# B&R Automation Studio project mappFramework (part 6)

#### HMIActions.st
```iecst
ACTION VC4_Init:

	brsmemset(ADR(HmiFile.Status.FifoSelect[0]), 0, SIZEOF(HmiFile.Status.FifoSelect));
	IF HmiFile.Parameters.Fifo.Enable THEN
		HmiFile.Status.FifoSelect[HmiFile.Parameters.Fifo.SelectedDevice] := 1;
	END_IF;

	HmiFile.Status.FIFOLayerStatus := HIDE;

END_ACTION

ACTION VC4_Cyclic:

	MpFileManagerUISys.MpLink := ADR(gMpLinkFileManagerUIFile);
	MpFileManagerUISys.UIConnect := ADR(MpFileManagerUIConnect);
	MpFileManagerUISys();

	FOR i := 0 TO ((SIZEOF(HmiFile.Status.FileNames)/SIZEOF(HmiFile.Status.FileNames[0])) - 1) DO
		HmiFile.Status.FileNames[i] := MpFileManagerUIConnect.File.List.Items[i].Name;

		// Time Stamp
		HmiFile.Status.TimeStamps[i] := DT_TO_STRING(MpFileManagerUIConnect.File.List.Items[i].LastModified);
		HmiFile.Status.TimeStamps[i] := RIGHT(HmiFile.Status.TimeStamps[i], 19);

		// File size
		HmiFile.Status.Size[i] := REAL_TO_STRING(UDINT_TO_REAL(MpFileManagerUIConnect.File.List.Items[i].Size) * 0.001);

		// Set image array based on item type
		IF MpFileManagerUIConnect.File.List.Items[i].IsFolder THEN
			HmiFile.Status.Type[i] := FOLDER;
		ELSIF NOT MpFileManagerUIConnect.File.List.Items[i].IsFolder AND MpFileManagerUIConnect.File.List.Items[i].IsSelected THEN
			HmiFile.Status.Type[i] := FILE_SELECTED;
		ELSE
			HmiFile.Status.Type[i] := FILE;
		END_IF

		// Fill file info string arrays
		IF MpFileManagerUIConnect.File.List.Items[i].IsFolder THEN
			HmiFile.Status.InfoFile.Type[i] := 'FOLDER';
		ELSE
			HmiFile.Status.InfoFile.Type[i] := 'FILE';
		END_IF
		IF MpFileManagerUIConnect.File.List.Items[i].IsSelected THEN
			HmiFile.Status.InfoFile.IsSelected[i] := '+';
		ELSE
			HmiFile.Status.InfoFile.IsSelected[i] := '-';
		END_IF

		// If file does not exist, clear objects
		IF HmiFile.Status.FileNames[i] = '' THEN
			HmiFile.Status.TimeStamps[i] := '';
			HmiFile.Status.Size[i] := '';
			HmiFile.Status.InfoFile.IsSelected[i] := '';
			HmiFile.Status.InfoFile.Type[i] := '';
		END_IF;

	END_FOR

	// Mutli selection
	IF (NOT MpFileManagerUIConnect.File.MultiSelect) THEN
		MpFileManagerUIConnect.File.List.Items[HmiFile.Status.SelectedIndex].IsSelected := TRUE;
	ELSIF (MpFileManagerUIConnect.File.MultiSelect) AND HmiFile.Commands.FileList.Clicked THEN
		MpFileManagerUIConnect.File.List.Items[HmiFile.Status.SelectedIndex].IsSelected := NOT MpFileManagerUIConnect.File.List.Items[HmiFile.Status.SelectedIndex].IsSelected;
	END_IF
	HmiFile.Commands.FileList.Clicked := FALSE;

	// Read currently selected device name for HMI
	IF (MpFileManagerUIConnect.DeviceList.SelectedIndex >= (SIZEOF(MpFileManagerUIConnect.DeviceList.DeviceNames) / SIZEOF(MpFileManagerUIConnect.DeviceList.DeviceNames[0]))) THEN
		MpFileManagerUIConnect.DeviceList.SelectedIndex := 0;
	END_IF
	HmiFile.Status.DeviceName := MpFileManagerUIConnect.DeviceList.DeviceNames[MpFileManagerUIConnect.DeviceList.SelectedIndex];

	// Read if current selected object is folder
	IF (HmiFile.Status.SelectedIndex >= (SIZEOF(MpFileManagerUIConnect.File.List.Items) / SIZEOF(MpFileManagerUIConnect.File.List.Items[0]))) THEN
		HmiFile.Status.SelectedIndex := 0;
	END_IF
	HmiFile.Status.IsFolder := MpFileManagerUIConnect.File.List.Items[HmiFile.Status.SelectedIndex].IsFolder;

	// Control the folder structure when entering and leaving folders
	IF (HmiFile.Commands.EnterFolder) AND MpFileManagerUIConnect.File.List.Items[HmiFile.Status.SelectedIndex].IsFolder THEN
		HmiFile.Commands.EnterFolder := FALSE;
		MpFileManagerUIConnect.File.EnterFolder := TRUE;
		FolderDepthCount := FolderDepthCount + 1;
	ELSE
		HmiFile.Commands.EnterFolder := FALSE;
	END_IF

	IF EDGEPOS(HmiFile.Commands.FolderUp) AND (HmiFile.Status.BackButton > 0) THEN
		HmiFile.Commands.FolderUp := FALSE;
		MpFileManagerUIConnect.File.FolderUp := TRUE;
		FolderDepthCount := FolderDepthCount - 1;
	END_IF

	HmiFile.Status.BackButton := (FolderDepthCount > 0);

	// File SelectedIndex manager
	IF HmiFile.Commands.FileList.PageUp THEN
		HmiFile.Commands.FileList.PageUp := FALSE;
		HmiFile.Status.SelectedIndex := 0;

	ELSIF HmiFile.Commands.FileList.PageDown THEN
		HmiFile.Commands.FileList.PageDown := FALSE;
		HmiFile.Status.SelectedIndex := ((SIZEOF(HmiFile.Status.FileNames)/SIZEOF(HmiFile.Status.FileNames[0])) - 1);

	ELSIF HmiFile.Commands.FileList.StepUp THEN
		HmiFile.Commands.FileList.StepUp := FALSE;
		IF HmiFile.Status.SelectedIndex <> 0 THEN
			HmiFile.Status.SelectedIndex := HmiFile.Status.SelectedIndex - 1;
		END_IF

	ELSIF HmiFile.Commands.FileList.StepDown THEN
		HmiFile.Commands.FileList.StepDown := FALSE;
		IF HmiFile.Status.SelectedIndex <> ((SIZEOF(HmiFile.Status.FileNames)/SIZEOF(HmiFile.Status.FileNames[0])) - 1) THEN
			HmiFile.Status.SelectedIndex := HmiFile.Status.SelectedIndex + 1;
		END_IF
	END_IF

	HmiFile.Status.DefaultFileSelected := ((MpFileManagerUIConnect.File.List.Items[HmiFile.Status.SelectedIndex].Name = 'Default.par') OR
		(MpFileManagerUIConnect.File.List.Items[HmiFile.Status.SelectedIndex].Name = 'Machine.mcfg')) AND
		MpFileManagerUIConnect.DeviceList.SelectedIndex = 0;

END_ACTION

ACTION FormatDeviceDataProvider:

	// Select CF device if USB device is not available
	FOR i := 0 TO IDX_USB_DEV_LIST DO
		tempIdx := (i + USBOffset);

		IF gUSBAvailable[i] THEN
			PathCheck.DeviceList.DeviceNames[tempIdx] := 'USB';
			brsitoa(i + 1, ADR(PathCheck.DeviceList.DeviceNames[tempIdx]) + brsstrlen(ADR(PathCheck.DeviceList.DeviceNames[tempIdx])));
		ELSE
			brsmemset(ADR(HmiFile.Status.DeviceDataProvider[tempIdx]), 0, SIZEOF(HmiFile.Status.DeviceDataProvider[tempIdx]));
			brsmemset(ADR(PathCheck.DeviceList.DeviceNames[tempIdx]), 0, SIZEOF(PathCheck.DeviceList.DeviceNames[tempIdx]));
		END_IF
	END_FOR

	MaxDeviceNameIndex := ((SIZEOF(MpFileManagerUIConnect.DeviceList.DeviceNames) / SIZEOF(MpFileManagerUIConnect.DeviceList.DeviceNames[0])) - 1);
	// Check initilized folder for existance and remove any from the device list that don't exist
	IF (IdentStatus = 0) THEN
		// Copy device name from source list into the actual device list
		MpFileManagerUIConnect.DeviceList.DeviceNames[Index] := PathCheck.DeviceList.DeviceNames[DeviceListCount];
		Index := Index + 1;
		DeviceListCount := DeviceListCount + 1;

		IF (DeviceListCount > ((SIZEOF(PathCheck.DeviceList.DeviceNames) / SIZEOF(PathCheck.DeviceList.DeviceNames[0])) - 1)) THEN
			DeviceListCount := 0;
		END_IF
		IF (Index > MaxDeviceNameIndex) THEN
			Index := 0;
		END_IF
	ELSIF (IdentStatus = 3324) THEN
		DeviceListCount := DeviceListCount + 1;
		IF DeviceListCount > ((SIZEOF(PathCheck.DeviceList.DeviceNames) / SIZEOF(PathCheck.DeviceList.DeviceNames[0])) - 1) THEN
			// Delete entries past the actual number of devices found
			FOR i:=Index TO MaxDeviceNameIndex DO
				MpFileManagerUIConnect.DeviceList.DeviceNames[i] := '';
			END_FOR
			DeviceListCount := 0;
			Index := 0;
		END_IF
	END_IF

	IdentStatus := ST_ident(ADR(PathCheck.PrgName[DeviceListCount]),0,ADR(Ident));

	// Create device data provider for FIFO drop down
	FOR i := 0 TO MaxDeviceNameIndex DO
		IF (MpFileManagerUIConnect.DeviceList.DeviceNames[i] <> '') THEN
			HmiFile.Status.DeviceDataProvider[i] := MpFileManagerUIConnect.DeviceList.DeviceNames[i];
		ELSE
			brsmemset(ADR(HmiFile.Status.DeviceDataProvider[i]), 0, SIZEOF(HmiFile.Status.DeviceDataProvider[i]));
		END_IF
	END_FOR

END_ACTION
```

### Package Logical/Infrastructure/VC4/Usb - Package for USB handling for mapp Framework

### Program Logical/Infrastructure/VC4/Usb/UsbMgr (IEC) - Sample for all AsUSB-Library-Functions

#### UsbMgr.st - Cyclic code
```iecst
//*********************************************************************************
// Copyright: B&R Industrial Automation GmbH
// Author: B&R Industrial Automation GmbH
// Created: April 12, 2022
// Description: This task automatically detects and (un)links USB storage devices
//*********************************************************************************

PROGRAM _INIT
END_PROGRAM

PROGRAM _CYCLIC

	CASE StateMachine OF
		// -----------------------------------------------------------------------------------------------------------
		// Wait state
		// -----------------------------------------------------------------------------------------------------------
		USB_WAIT:
			// Refresh USB data every X seconds when enabled
			Node := 1;
			USB.Status := ERR_OK;
			IF USB.Cmd.AutoScan THEN
				RefreshTimer(IN := 1, PT := USB.Par.RefreshInterval);
				// Get new USB data
				IF(RefreshTimer.Q) THEN
					RefreshTimer(IN := 0);
					USB.Status := ERR_FUB_BUSY;
					brsmemset(ADR(UsbData), 0, SIZEOF(UsbData));
					StateMachine := USB_CREATE_NODE_ID_LIST;
				END_IF
			ELSE
				RefreshTimer(IN := 0);
			END_IF
			// Refresh USB data every X seconds when enabled
			IF USB.Cmd.ErrorReset THEN
				StateMachine := USB_ERROR;
			END_IF

			FOR i := 0 TO IDX_USB_DEV_LIST DO
				gUSBAvailable[i] := USB.Par.IsConnected[i+1];
			END_FOR

			// -----------------------------------------------------------------------------------------------------------
			// Get USB device list
			// -----------------------------------------------------------------------------------------------------------
		USB_CREATE_NODE_ID_LIST:
			GetUsbNodeList.enable := 1;
			GetUsbNodeList.pBuffer := ADR(NodeIdBuffer);
			GetUsbNodeList.bufferSize := SIZEOF(NodeIdBuffer);
			GetUsbNodeList.filterInterfaceClass := asusb_CLASS_MASS_STORAGE;
			GetUsbNodeList.filterInterfaceSubClass := 0;
			GetUsbNodeList;

			// --------------------------------------------------------------------------------------------------------------------
			// Success
			IF GetUsbNodeList.status = 0 THEN
				StateMachine := USB_READ_DEVICE_DATA;
				Node := 1;
				// No USB devices found
			ELSIF GetUsbNodeList.status = asusbERR_USB_NOTFOUND THEN
				// Unlink old device if it is gone now otherwise wait for next round
				FOR i:=1 TO MAX_IDX_USB_DEV_LIST DO
					IF(USB.Par.IsConnected[i]) THEN
						Node := 1;
						StateMachine := USB_CHECK_LINKED;
						RETURN;
					END_IF
				END_FOR;
				StateMachine := USB_WAIT;
				// Error
			ELSIF GetUsbNodeList.status <> ERR_FUB_BUSY THEN
				USB.Status := GetUsbNodeList.status;
				USB.Err.State := StateMachine;
				IF GetUsbNodeList.status = asusbERR_BUFSIZE THEN
					USB.Err.Text := 'maximum number of devices reached';
				ELSE
					USB.Err.Text := 'error getting device list';
				END_IF;
				StateMachine := USB_ERROR;
			END_IF;
			// -----------------------------------------------------------------------------------------------------------
			// Get device information
			// -----------------------------------------------------------------------------------------------------------
		USB_READ_DEVICE_DATA:
			GetUsbNode.enable := 1;
			GetUsbNode.nodeId := NodeIdBuffer[Node];
			GetUsbNode.pBuffer := ADR(UsbData[Node]);
			GetUsbNode.bufferSize := SIZEOF (UsbData[Node]);
			GetUsbNode;

			// --------------------------------------------------------------------------------------------------------------------
			// Success
			IF GetUsbNode.status = 0 THEN
				// Make sure we have enough space to store USB data, proceed with next StateMachine when all devices are detetced
				IF (Node = GetUsbNodeList.listNodes) OR (Node = MAX_IDX_USB_DEV_LIST) THEN
					Node := 1;
					StateMachine := USB_CHECK_LINKED;
					// Get next USB device
				ELSE
					Node := Node + 1;
				END_IF;
				// Error
			ELSIF GetUsbNode.status <> ERR_FUB_BUSY THEN
				USB.Status := GetUsbNode.status;
				USB.Err.State := StateMachine;
				USB.Err.Text := 'error getting device data';
				StateMachine := USB_ERROR;
			END_IF;
			// -----------------------------------------------------------------------------------------------------------
			// Check if linked device are still present
			// -----------------------------------------------------------------------------------------------------------
		USB_CHECK_LINKED:
			// Proceed to new devices when last device was checked
			IF(Node > MAX_IDX_USB_DEV_LIST) THEN
				Node := 1;
				StateMachine := USB_LINK_NEW;
				RETURN;
			END_IF

			// -----------------------------------------------------------------------------------------------------------
			// Check if device is still active
			IsLinked := FALSE;
			FOR i:=1 TO MAX_IDX_USB_DEV_LIST DO
				// Compare old and new data
				IF(brsmemcmp(ADR(UsbDataOld[Node]), ADR(UsbData[i]), SIZEOF(UsbData[i])) = 0) AND
					((NOT USB.Par.IgnoreDongle) OR (USB.Par.IgnoreDongle AND UsbData[i].productId <> BrProductId AND UsbData[i].vendorId <> BrVendorId)) THEN
					// Clear data, mark as linked and EXIT loop
					brsmemset(ADR(UsbData[i]), 0, SIZEOF(UsbData[i]));
					IsLinked := TRUE;
					EXIT;
				END_IF
			END_FOR;

			// -----------------------------------------------------------------------------------------------------------
			// Find next linked device
			IF(IsLinked OR UsbDataOld[Node].interfaceClass = 0) THEN
				IF(Node < MAX_IDX_USB_DEV_LIST) THEN
					Node := Node + 1;
					WHILE(Node < MAX_IDX_USB_DEV_LIST AND UsbDataOld[Node].interfaceClass = 0) DO
						Node := Node + 1;
					END_WHILE;
					IF(Node = MAX_IDX_USB_DEV_LIST AND UsbDataOld[Node].interfaceClass = 0) THEN
						Node := Node + 1;
					END_IF
				ELSE
					Node := Node + 1;
				END_IF
				// Unlink device if it is missing
			ELSE
				StateMachine := USB_UNLINK_DEVICE;
			END_IF
			// -----------------------------------------------------------------------------------------------------------
			// Link new devices
			// -----------------------------------------------------------------------------------------------------------
		USB_LINK_NEW:
			// Return to wait state when last device was checked
			IF(Node > MAX_IDX_USB_DEV_LIST) THEN
				StateMachine := USB_WAIT;
				RETURN;
			END_IF

			// -----------------------------------------------------------------------------------------------------------
			// Find next new device
			IF(UsbData[Node].interfaceClass <> 0) THEN
				IF((NOT USB.Par.IgnoreDongle) OR (UsbData[Node].productId <> BrProductId AND UsbData[Node].vendorId <> BrVendorId)) THEN
					StateMachine := USB_LINK_DEVICE;
					RETURN;
				END_IF
			END_IF
			Node := Node + 1;
			// -----------------------------------------------------------------------------------------------------------
			// Link device
			// -----------------------------------------------------------------------------------------------------------
		USB_LINK_DEVICE:
			// Find empty slot
			FOR i:=1 TO MAX_IDX_USB_DEV_LIST DO
				IF(UsbDataOld[i].interfaceClass = 0) THEN
					EXIT;
				END_IF
			END_FOR;
			// No more slot available
			IF(i = MAX_IDX_USB_DEV_LIST AND UsbDataOld[i].interfaceClass <> 0) THEN
				USB.Status := ERR_MAX_DEVICE;
				USB.Err.State := StateMachine;
				USB.Err.Text := 'maximum number of device reached';
				StateMachine := USB_ERROR;
				RETURN;
			END_IF
			// Create device string
			brsstrcpy(ADR(DevicePara), ADR('/DEVICE='));
			brsstrcat(ADR(DevicePara), ADR(UsbData[Node].ifName));
			brsstrcpy(ADR(DeviceName), ADR('USB'));
			brsitoa(i, ADR(tmpSTR));
			brsstrcat(ADR(DeviceName), ADR(tmpSTR));
			// Link device
			DevLinkSys.enable := 1;
			DevLinkSys.pDevice := ADR(DeviceName);
			DevLinkSys.pParam := ADR(DevicePara);
			DevLinkSys;

			// --------------------------------------------------------------------------------------------------------------------
			// Success
			IF DevLinkSys.status = 0 THEN
				// Store data for new device
				brsmemcpy(ADR(UsbDataOld[i]), ADR(UsbData[Node]), SIZEOF(UsbData[Node]));
				USB.Par.IsConnected[i] := TRUE;
				LinkHandle[i] := DevLinkSys.handle;
				Node := Node + 1;
				StateMachine := USB_LINK_NEW;
				// Error
			ELSIF DevLinkSys.status <> ERR_FUB_BUSY THEN
				USB.Status := DevLinkSys.status;
				USB.Err.State := StateMachine;
				USB.Err.Text := 'error linking device';
				StateMachine := USB_ERROR;
			END_IF;
			// -----------------------------------------------------------------------------------------------------------
			// UnLink device
			// -----------------------------------------------------------------------------------------------------------
		USB_UNLINK_DEVICE:
			DevUnlinkSys.enable := 1;
			DevUnlinkSys.handle := LinkHandle[Node];
			DevUnlinkSys;

			// --------------------------------------------------------------------------------------------------------------------
			// Success
			IF DevUnlinkSys.status = 0 THEN
				// Clear data
				brsmemset(ADR(UsbDataOld[Node]), 0, SIZEOF(UsbDataOld[Node]));
				USB.Par.IsConnected[Node] := FALSE;
				LinkHandle[Node] := 0;
				// Find next linked device
				WHILE(Node < MAX_IDX_USB_DEV_LIST AND UsbDataOld[Node].interfaceClass = 0) DO
					Node := Node + 1;
				END_WHILE;
				IF(Node = MAX_IDX_USB_DEV_LIST AND UsbDataOld[Node].interfaceClass = 0) THEN
					Node := Node + 1;
				END_IF
				StateMachine := USB_CHECK_LINKED;
				// Error
			ELSIF DevUnlinkSys.status <> ERR_FUB_BUSY THEN
				// Clear data
				brsmemset(ADR(UsbDataOld[Node]), 0, SIZEOF(UsbDataOld[Node]));
				USB.Par.IsConnected[Node] := FALSE;
				LinkHandle[Node] := 0;

				brsitoa(Node, ADR(tmpSTR));
				USB.Status := DevUnlinkSys.status;
				USB.Err.State := StateMachine;
				USB.Err.Text := 'error unlinking device no ';
				brsstrcat(ADR(USB.Err.Text), ADR(tmpSTR));
				StateMachine := USB_ERROR;
			END_IF;
			// -----------------------------------------------------------------------------------------------------------
			// Error state
			// -----------------------------------------------------------------------------------------------------------
		USB_ERROR:
			// Get more error information
			IF(USB.Status = 0) THEN
				USB.Status := FileIoGetSysError();
			END_IF

			// Unlink device
			IF(USB.Err.State = USB_LINK_DEVICE) THEN
				DevUnlinkSys.enable := 1;
				DevUnlinkSys.handle := DevLinkSys.handle;
				DevUnlinkSys;
			END_IF

			// Reset error
			IF(USB.Cmd.ErrorReset AND DevUnlinkSys.status <> ERR_FUB_BUSY) THEN
				USB.Cmd.ErrorReset := FALSE;
				brsmemset(ADR(USB.Err), 0, SIZEOF(USB.Err));
				StateMachine := USB_WAIT;
			END_IF
	END_CASE;

END_PROGRAM

PROGRAM _EXIT
	FOR i:=1 TO MAX_IDX_USB_DEV_LIST DO
		REPEAT
			DevUnlinkSys.enable := 1;
			DevUnlinkSys.handle := LinkHandle[i];
			DevUnlinkSys;
			UNTIL DevUnlinkSys.status <> ERR_FUB_BUSY
		END_REPEAT;
	END_FOR;
END_PROGRAM
```

#### UsbMgr.typ - Local data types
```iecst
TYPE
	UsbStateEnum :
		(
		USB_WAIT, (*Wait for starting the Function chain*)
		USB_CREATE_NODE_ID_LIST, (*Create a list of Node-IDs from all active USB devices*)
		USB_READ_DEVICE_DATA, (*Read out the specific data from the Node-IDs*)
		USB_CHECK_LINKED, (*Check if device is still connected*)
		USB_LINK_NEW,
		USB_LINK_DEVICE, (*Link file device*)
		USB_UNLINK_DEVICE, (*Unlink the File Device from specific path*)
		USB_ERROR (*Jump to this step in every case of Error occuring in the Function chain*)
		);
	UsbCmdType : 	STRUCT
		AutoScan : BOOL := TRUE; (*Scan USB ports automatically*)
		ErrorReset : BOOL; (*Reset error*)
	END_STRUCT;
	UsbParType : 	STRUCT
		IgnoreDongle : BOOL := TRUE; (*Ignoe B&R license dongle*)
		RefreshInterval : TIME := T#3s; (*Intervall timer for USB device refresh*)
		IsConnected : ARRAY[0..MAX_IDX_USB_DEV_LIST]OF BOOL; (*Shows if a USB stick is connected*)
	END_STRUCT;
	UsbErrType : 	STRUCT
		State : UsbStateEnum; (*State where the error occured*)
		Text : STRING[80]; (*Error text*)
	END_STRUCT;
	UsbMainType : 	STRUCT
		Cmd : UsbCmdType; (*Command structure*)
		Par : UsbParType; (*Parameter structure*)
		Err : UsbErrType; (*Error structure*)
		Status : UINT; (*Current status*)
	END_STRUCT;
END_TYPE
```

#### UsbMgr.var - Local variables
```iecst
(*Function Blocks*)
VAR
	RefreshTimer : TON;
	GetUsbNodeList : UsbNodeListGet; (*Type of FUB UsbNodeListGet*)
	GetUsbNode : UsbNodeGet; (*Type of FUB UsbNodeGet*)
	DevLinkSys : DevLink; (*Type of FUB DevLink*)
	DevUnlinkSys : DevUnlink; (*Type of FUB DevUnlink*)
END_VAR
(*Constants*)
VAR CONSTANT
	BrVendorId : UINT := 1615; (*B&R vendor id*)
	BrProductId : UINT := 1001; (*B&R dongle product id*)
END_VAR
(*Structure Types*)
VAR
	USB : UsbMainType;
	StateMachine : UsbStateEnum; (*State machine*)
	UsbData : ARRAY[1..MAX_IDX_USB_DEV_LIST] OF usbNode_typ; (*Data of all available USB devices*)
	UsbDataOld : ARRAY[1..MAX_IDX_USB_DEV_LIST] OF usbNode_typ; (*Old data of all available USB devices*)
END_VAR
(*Variables*)
VAR
	DevicePara : STRING[80]; (*Connection path of USB device*)
	DeviceName : STRING[40]; (*Connection path of USB device*)
	LinkHandle : ARRAY[1..MAX_IDX_USB_DEV_LIST] OF UDINT; (*Link handle for USB device*)
	NodeIdBuffer : ARRAY[1..MAX_IDX_USB_DEV_LIST] OF UDINT; (*Different nodeIDs saved in array-elements*)
	IsLinked : BOOL; (*Helper variable that indicates that a USB stick is linked*)
	Node : USINT; (*Node number*)
	i : USINT;
	tmpSTR : STRING[10];
	ERR_MAX_DEVICE : UINT := 50000; (*Maximum number of dongles reached*)
END_VAR
```

### Package Logical/Infrastructure/VC4/Recipe - Package for mapp Recipe Framework

### Program Logical/Infrastructure/VC4/Recipe/RecipeMgr (IEC)

#### RecipeMgr.st - Init, cyclic, exit code
```iecst
//***********************************************************************
// Copyright: B&R Industrial Automation GmbH
// Author: B&R Industrial Automation GmbH
// Created: Jan 1, 2022
// Description: Tasks for recipe control with VC4 front-end.
//***********************************************************************

PROGRAM _INIT

	// Create folder for this component on the user file device
	DirCreateRecipe(enable := TRUE, pDevice := ADR('mappRecipeFiles'), pName := ADR('/'));

	// Wait for DirCreate_0 to complete.
	WHILE (DirCreateRecipe.status = ERR_FUB_BUSY) DO
		DirCreateRecipe();
	END_WHILE

	// Check if folder already exist and if so disabled the function block call
	IF DirCreateRecipe.status = fiERR_DIR_ALREADY_EXIST OR (DirCreateRecipe.status = ERR_OK) THEN
		DirCreateRecipe(enable := FALSE);
	END_IF

	// Initialize mapp function blocks
	// By default, the Framework sets up an XML recipe system. To swtich to the CSV format, refer to the "Change Recipe Format"
	// page in the AS Help (GUID 2052b3a5-f59b-45f9-9fcd-3289c93401af)
	MpRecipeUISetup.Confirmation.RecipeDelete := TRUE;
	MpRecipeUISetup.RecipeListSize := 9;
	MpRecipeUISetup.RecipeListScrollWindow := 0;
	MpRecipeUISetup.AutoLoadHeader := TRUE;
	MpRecipeUIConnect.New.FileName := 'newRecipe';
	MpRecipeUIConnect.Recipe.Filter := '*par';
	MpRecipeUISys.MpLink := ADR(gMpLinkRecipeXml);
	MpRecipeUISys.Enable := TRUE;
	MpRecipeUISys.UIConnect := ADR(MpRecipeUIConnect);
	MpRecipeUISys.UISetup := MpRecipeUISetup;
	MpRecipeUISys();

	HmiRecipe.Parameters.Category := PARAMETERS_CATEGORY;
	HmiRecipe.Status.DeviceDataProvider[0] := '{"value":"mappRecipeFiles","text":"CF/PLC"}';
	HmiRecipe.Parameters.DeviceName := 'mappRecipeFiles';
	MpRecipeSys.MpLink := ADR(gMpLinkRecipeXml);
	MpRecipeSys.Enable := TRUE;
	MpRecipeSys.Category := ADR(HmiRecipe.Parameters.Category);
	MpRecipeSys.DeviceName := ADR(HmiRecipe.Parameters.DeviceName);
	MpRecipeSys.FileName := ADR(HmiRecipe.Parameters.FileName);
	MpRecipeSys.Header := ADR(Header);

	// Wait for MpRecipeSys to activate. This must be active before you can call the RegPar function blocks, which is below.
	WHILE NOT(MpRecipeSys.Active OR MpRecipeSys.Error) DO
		MpRecipeSys();
	END_WHILE

	// Register the preview variables to the recipe. These preview variables are a buffer between the recipe system and the
	// variables used at runtime on the machine (Parameters, MachineSettings). By using these preview variables, you can
	// preview and edit a recipe on the HMI without actually loading it to the machine. For more details, refer to the
	// "Recipe System Design" page in the AS Help (GUID 3ccd7409-0b52-4bbc-a93a-4010f6db414c).

	MpRecipeRegPar_PreviewPar.MpLink := ADR(gMpLinkRecipeXml);
	MpRecipeRegPar_PreviewPar.Enable := TRUE;
	MpRecipeRegPar_PreviewPar.PVName := ADR('RecipeMgr:ParametersPreview');
	MpRecipeRegPar_PreviewPar.Category := ADR(PARAMETERS_CATEGORY);
	MpRecipeRegPar_PreviewPar();

	MpRecipeRegPar_PreviewCfg.MpLink := ADR(gMpLinkRecipeXml);
	MpRecipeRegPar_PreviewCfg.Enable := TRUE;
	MpRecipeRegPar_PreviewCfg.PVName := ADR('RecipeMgr:MachineSettingsPreview');
	MpRecipeRegPar_PreviewCfg.Category := ADR(MACHINE_CONFIGURATION_CATEGORY);
	MpRecipeRegPar_PreviewCfg();

	// Wait for RegPar function blocks to activate. These must be active before you can load a recipe,
	// which is further down in the Initialization program.
	WHILE NOT(MpRecipeRegPar_PreviewPar.Active OR MpRecipeRegPar_PreviewPar.Error) DO
		MpRecipeRegPar_PreviewPar();
	END_WHILE
	WHILE NOT(MpRecipeRegPar_PreviewCfg.Active OR MpRecipeRegPar_PreviewCfg.Error) DO
		MpRecipeRegPar_PreviewCfg();
	END_WHILE

	// Load default Machine Settings recipe
	HmiRecipe.Parameters.Category := MACHINE_CONFIGURATION_CATEGORY;
	HmiRecipe.Parameters.FileName := DEFAULT_MACHINE_CONFIGURATION;
	brsstrcat(ADR(HmiRecipe.Parameters.FileName),ADR(MACHINE_CONFIG_FILE_EXTENSION));
	MpRecipeSys.Load := TRUE;
	WHILE NOT(MpRecipeSys.CommandDone OR MpRecipeSys.Error) DO
		MpRecipeSys();
	END_WHILE
	MachineSettings := MachineSettingsPreview;
	HmiRecipe.Status.LastLoadedConfigRecipe := DEFAULT_MACHINE_CONFIGURATION;
	brsstrcat(ADR(HmiRecipe.Status.LastLoadedConfigRecipe),ADR(MACHINE_CONFIG_FILE_EXTENSION));
	HmiRecipe.Status.ConfigRecipeLoaded := TRUE;

	// Check if the default machine settings recipe is missing
	IF MpRecipeSys.Info.Diag.StatusID.ID = mpRECIPE_ERR_LOAD_DATA THEN
		HmiRecipe.Status.MachineSettingsRecipeMissing := TRUE;
		HmiRecipe.Status.LastLoadedConfigRecipe := '';
		HmiRecipe.Status.ConfigRecipeLoaded := FALSE;
	END_IF

	MpRecipeSys.ErrorReset := MpRecipeSys.Error;
	MpRecipeSys.Load := FALSE;
	MpRecipeSys();

	// Load default Parameter recipe
	HmiRecipe.Parameters.Category := PARAMETERS_CATEGORY;
	HmiRecipe.Parameters.FileName := DEFAULT_PARAMETERS;
	brsstrcat(ADR(HmiRecipe.Parameters.FileName),ADR(PARAMETERS_FILE_EXTENSION));
	HmiRecipe.Status.PreviousRecipe := DEFAULT_PARAMETERS;
	MpRecipeSys.Load := TRUE;
	WHILE NOT(MpRecipeSys.CommandDone OR MpRecipeSys.Error) DO
		MpRecipeSys();
	END_WHILE
	Parameters := ParametersPreview;
	HmiRecipe.Status.LastLoadedProductRecipe := DEFAULT_PARAMETERS;
	brsstrcat(ADR(HmiRecipe.Status.LastLoadedProductRecipe),ADR(PARAMETERS_FILE_EXTENSION));
	HmiRecipe.Status.ProductRecipeLoaded := TRUE;

	// Check if the default parameters recipe is missing
	IF MpRecipeSys.Info.Diag.StatusID.ID = mpRECIPE_ERR_LOAD_DATA THEN
		HmiRecipe.Status.ParameterRecipeMissing := TRUE;
		HmiRecipe.Status.LastLoadedProductRecipe := '';
		HmiRecipe.Status.ProductRecipeLoaded := FALSE;
	END_IF

	MpRecipeSys.ErrorReset := MpRecipeSys.Error;
	MpRecipeSys.Load := FALSE;
	MpRecipeSys();

	// Trigger update notification so that the initial parameters are copied to the process
	MpRecipeSys.UpdateNotification := TRUE;

	// Init Filemanager for exporting/importing files
	MpFileManagerUIRecipe.Enable := TRUE;
	MpFileManagerUIRecipe.MpLink := ADR(gMpLinkFileManagerUIRecipe);
	MpFileManagerUIRecipe.UIConnect := ADR(MpFileManagerUIConnect);
	MpFileManagerUIRecipe.UISetup.FileListSize := SIZEOF(MpFileManagerUIConnect.File.List.Items) / SIZEOF(MpFileManagerUIConnect.File.List.Items[0]);
	MpFileManagerUIConnect.DeviceList.DeviceNames[0] := 'mappRecipeFiles';
	MpFileManagerUIConnect.DeviceList.DeviceNames[1] := '';
	MpFileManagerUIRecipe();

	HmiRecipe.Status.HMIcommand := REC_HMI_WAIT;

	VC4_Init;

END_PROGRAM

PROGRAM _CYCLIC

	// Call actions
	FormatDeviceDataProvider;
	LoadPreview;
	RecipeHMIcommands;
	LoadStatus;

	// Reset commands on MpRecipe FUB
	IF MpRecipeSys.CommandDone THEN
		MpRecipeSys.Load := FALSE;
		MpRecipeSys.Save := FALSE;
		// Set update notification for machine category
		IF ((brsstrcmp(ADR(HmiRecipe.Parameters.Category), ADR(MACHINE_CONFIGURATION_CATEGORY)) = 0) AND (MpRecipeSys.Save)) THEN
			MpRecipeSys.UpdateNotification := TRUE;
		ELSE
			MpRecipeSys.UpdateNotification := FALSE;
		END_IF
	END_IF

	// Error reset
	IF NOT MpRecipeSys.Error THEN
		MpRecipeSys.ErrorReset := FALSE;
	END_IF

	IF NOT MpRecipeUISys.Error THEN
		MpRecipeUISys.ErrorReset := FALSE;
	END_IF

	// Assign MpLinks & address references
	MpRecipeSys.MpLink := ADR(gMpLinkRecipeXml);
	MpRecipeSys.DeviceName := ADR(HmiRecipe.Parameters.DeviceName);
	MpRecipeSys.Header := ADR(Header);
	MpRecipeUISys.MpLink := ADR(gMpLinkRecipeXml);
	MpRecipeUISys.UIConnect := ADR(MpRecipeUIConnect);
	MpFileManagerUIRecipe.MpLink := ADR(gMpLinkFileManagerUIRecipe);
	MpRecipeRegPar_PreviewPar.MpLink := ADR(gMpLinkRecipeXml);
	MpRecipeRegPar_PreviewPar.PVName := ADR('RecipeMgr:ParametersPreview');
	MpRecipeRegPar_PreviewPar.Category := ADR(PARAMETERS_CATEGORY);
	MpRecipeRegPar_PreviewCfg.MpLink := ADR(gMpLinkRecipeXml);
	MpRecipeRegPar_PreviewCfg.PVName := ADR('RecipeMgr:MachineSettingsPreview');
	MpRecipeRegPar_PreviewCfg.Category := ADR(MACHINE_CONFIGURATION_CATEGORY);
	MpFileManagerUIRecipe.UIConnect := ADR(MpFileManagerUIConnect);

	// Call function blocks
	MpRecipeSys();
	MpRecipeUISys();
	MpFileManagerUIRecipe();
	MpRecipeRegPar_PreviewPar();
	MpRecipeRegPar_PreviewCfg();

END_PROGRAM

PROGRAM _EXIT

	// Disable the function blocls to unlink the MpLinks
	MpRecipeSys.Enable := FALSE;
	MpRecipeUISys.Enable := FALSE;
	MpRecipeRegPar_PreviewPar.Enable := FALSE;
	MpRecipeRegPar_PreviewCfg.Enable := FALSE;
	MpFileManagerUIRecipe.Enable := FALSE;

	// Call function blocks
	MpRecipeSys();
	MpRecipeUISys();
	MpRecipeRegPar_PreviewPar();
	MpRecipeRegPar_PreviewCfg();
	MpFileManagerUIRecipe();

END_PROGRAM
```

#### RecipeMgr.typ - Local data types
```iecst
(*Structure types*)

TYPE
	RecipeHmiInterfaceType : 	STRUCT  (*Structure to hold commands, parameters and status from the HMI*)
		Commands : RecipeCommandsType; (*Structure to hold the commands from the HMI*)
		Parameters : RecipeParametersType; (*Structure to hold the parameters for the HMI*)
		Status : RecipeStatusType; (*Structure to hold status information from the mapp View HMI*)
	END_STRUCT;
	RecipeCommandsType : 	STRUCT  (*Structure to hold the commands from the HMI*)
		LoadRecipe : BOOL; (*Load recipe*)
		SaveSelectedRecipe : BOOL; (*Save the selected recipe (which is not necessarily the active recipe)*)
		CreateRecipe : BOOL; (*Create recipe*)
		ImportFromUSB : BOOL; (*Import from USB device*)
		ExportToUSB : BOOL; (*Export to USB device*)
		ResetPreview : BOOL; (*Reset the preview to empty/zeros in the event of an invalid recipe*)
	END_STRUCT;
	RecipeParametersType : 	STRUCT  (*Structure to hold the parameters for the HMI*)
		Category : STRING[30]; (*Current category*)
		CategoryIndex : USINT; (*Current category*)
		DeviceName : STRING[50]; (*Selected file device name*)
		FileName : STRING[255]; (*Recipe file name*)
	END_STRUCT;
	RecipeStatusType : 	STRUCT  (*Structure to hold status information from the mapp View HMI*)
		DefaultFilesDeleteButtonStatus : USINT;
		HMIcommand : RecipeHmiStepEnum; (*State machine step for HMI commands*)
		LastLoadedConfigRecipe : STRING[255]; (*Last loaded configuration recipe*)
		LastLoadedProductRecipe : STRING[255]; (*Last loaded product recipe*)
		ProductRecipeLoaded : BOOL; (*Product recipe was loaded*)
		ConfigRecipeLoaded : BOOL; (*Config recipe was loaded*)
		LastMaxSelection : UINT; (*The previous maximum number of recipes*)
		LastSelectedIndex : UINT; (*The previous selected index*)
		LastStatus : MpRecipeUIStatusEnum; (*The previous UI status*)
		EditDialogOpened : BOOL; (*Flag that the edit dialog box was opened*)
		CreateDialogOpened : BOOL; (*Flag that the create dialog box was opened*)
		PreviousRecipe : STRING[80]; (*Name of the previous recipe*)
		FileDuplicate : BOOL; (*Recipe file already exists, warn the user.*)
		FilesAvailable : BOOL; (*Control access to widget when no files are available*)
		InvalidRecipe : BOOL; (*The selected recipe cannot be previewed*)
		LoadingRecipeList : BOOL; (*The recipe list is loading*)
		MachineSettingsRecipeMissing : BOOL; (*Flag for if the default machine settings recipe is not present*)
		ParameterRecipeMissing : BOOL; (*Flag for if the default parameters recipe is not present*)
		LoadAllowed : BOOL; (*Flag for whether you can load a recipe. Recipe must exist and be valid. *)
		DeviceDataProvider : ARRAY[0..MAX_IDX_FILE_DEV]OF STRING[100]; (*File device data provider*)
		SelectedRecipe : STRING[255]; (*The name of the selected recipe*)
		ActiveRecipe : STRING[255];
		DefaultRecipeLayer : RecipeStatusDefRecLayerType;
		CreateRecipeLayer : RecipeStatusCteateRecLayerType;
		PreviewRecipeLayer : RecipeStatusPreviewRecLayerType;
		RecipeLoadLayer : RecipeStatusRecipeLoadLayerType;
		EditRecipeLayer : RecipeStatusEditRecLayerType;
		DuplicateLayer : USINT;
		DeviceValid : BOOL; (*Flag for whether FileDevice is valid. Prevents user from being prompted to load default recipe.*)
		InvalidRecipeLayer : BOOL;
		DefaultFilesCannotBeDeleteLayer : USINT;
		RecipePageOpenedNow : BOOL;
		LoadPreviewAfterPageOpened : BOOL;
	END_STRUCT;
	RecipeStatusDefRecLayerType : 	STRUCT
		Status : USINT;
	END_STRUCT;
	RecipeStatusCteateRecLayerType : 	STRUCT
		ParsStatus : USINT;
		MachConfigStatus : USINT;
		FileNameInputActive : USINT;
	END_STRUCT;
	RecipeStatusPreviewRecLayerType : 	STRUCT
		ParsStatus : USINT;
		MachConfigStatus : USINT;
	END_STRUCT;
	RecipeStatusRecipeLoadLayerType : 	STRUCT
		Status : USINT;
	END_STRUCT;
	RecipeStatusEditRecLayerType : 	STRUCT
		ParsStatus : USINT;
		MachConfigStatus : USINT;
		Save : BOOL;
	END_STRUCT;
	ParametersType : 	STRUCT  (*Demo / starter structure for machine parameters*)
		AddParametersHere1 : BOOL; (*Add your parameteres here *)
		AddParametersHere2 : STRING[80]; (*Add your parameteres here *)
		AddParametersHere3 : REAL; (*Add your parameteres here *)
		AddParametersHere4 : REAL; (*Add your parameteres here *)
		AddParametersHere5 : REAL; (*Add your parameteres here *)
	END_STRUCT;
	MachineSettingsType : 	STRUCT  (*Demo / starter structure for machine configuration settings*)
		AddMachineSettingsHere1 : USINT; (*Add your settings here*)
		AddMachineSettingsHere2 : DINT; (*Add your settings here*)
		AddMachineSettingsHere3 : BOOL; (*Add your settings here*)
		AddMachineSettingsHere4 : REAL; (*Add your settings here*)
		AddMachineSettingsHere5 : UINT; (*Add your settings here*)
	END_STRUCT;
END_TYPE

(*Enumerations*)

TYPE
	RecipeHmiStepEnum :
		( (*State machine step for HMI commands*)
		REC_HMI_WAIT, (*Wait*)
		REC_HMI_LOAD, (*Load recipe*)
		REC_HMI_SAVE, (*Save recipe*)
		REC_HMI_CREATE, (*Create recipe*)
		REC_HMI_RESET_PREVIEW (*Reset the preview values to 0 / empty*)
		);
END_TYPE

(**)
```

#### RecipeMgr.var - Local variables
```iecst
(*Function Blocks*)
VAR
	MpRecipeSys : MpRecipeXml; (*MpRecipe instance*)
	MpRecipeRegPar_PreviewPar : MpRecipeRegPar; (*MpRecipeRegPar instance for ParametersPreview variable*)
	MpRecipeRegPar_PreviewCfg : MpRecipeRegPar; (*MpRecipeRegPar instance for MachineSettingsPreview*)
	MpRecipeUISys : MpRecipeUI; (*MpRecupeUI instance*)
	MpFileManagerUIRecipe : MpFileManagerUI; (*MpFileManagerUI instance*)
	DTGetTimeRecipe : DTGetTime; (*DTGetTime instance*)
	DirCreateRecipe : DirCreate; (*DirCreate instance*)
END_VAR
(*Constants*)
VAR CONSTANT
	MAX_IDX_FILE_DEV : USINT := MAX_IDX_USB_DEV_LIST + 1; (*Maximum number of  file devices *)
END_VAR
VAR
	PARAMETERS_RECIPE : STRING[50] := 'Parameters'; (*Value of the DropDownBox selection for the Parameters category*)
	MACHINE_CONFIGURATION_RECIPE : STRING[50] := 'Machine Configuration'; (*Value of the DropDownBox selection for the Machine Configuration category*)
END_VAR
(*Structure Types*)
VAR
	HmiRecipe : RecipeHmiInterfaceType; (*HMI interface structure*)
	Parameters : ParametersType; (*Machine parameters. Used by the machine at runtime*)
	ParametersEdit : {REDUND_UNREPLICABLE} ParametersType; (*Machine parameters edit structure. Enables you to edit a recipe that is not currently active*)
	ParametersPreview : ParametersType; (*Machine parameters preview structure. Registered to the recipe. Enables you to preview a recipe that is not currently active.*)
	MachineSettings : MachineSettingsType; (*Machine settings. Used by the machine at runtime.*)
	MachineSettingsEdit : MachineSettingsType; (*Machine settings edit structure. Enables you to edit a recipe that is not currently active*)
	MachineSettingsPreview : MachineSettingsType; (*Machine settings preview structure. Registered to the recipe. Enables you to preview a recipe that is not currently active. *)
	MpRecipeUIConnect : MpRecipeUIConnectType; (*MpRecipeUI connection to the HMI*) (*ParameterFileStep : INT;*)
	MpRecipeUISetup : MpRecipeUISetupType; (*MpRecipeUI setup connection to the HMI*) (*ParameterFileStep : INT;*)
	MpFileManagerUIConnect : MpFileManagerUIConnectType; (*File manager connection to the HMI*)
	Header : MpRecipeXmlHeaderType; (*Header information*)
END_VAR
(*Variables*)
VAR
	i : USINT; (*Index to loop through file devices*)
	temp : STRING[260]; (*Temporary recipe name, used to check for duplicates when creating a new recipe*)
END_VAR
```

#### HMIActions.st - Supporting code for the HMI interface
```iecst
ACTION VC4_Init:

	HmiRecipe.Status.CreateRecipeLayer.ParsStatus			:= HIDE;
	HmiRecipe.Status.CreateRecipeLayer.MachConfigStatus		:= HIDE;
	HmiRecipe.Status.DefaultRecipeLayer.Status				:= HIDE;
	HmiRecipe.Status.RecipeLoadLayer.Status					:= HIDE;
	HmiRecipe.Status.EditRecipeLayer.ParsStatus				:= HIDE;
	HmiRecipe.Status.EditRecipeLayer.MachConfigStatus		:= HIDE;
	HmiRecipe.Status.DuplicateLayer							:= HIDE;
	HmiRecipe.Status.DefaultFilesCannotBeDeleteLayer		:= HIDE;
	HmiRecipe.Status.CreateRecipeLayer.FileNameInputActive	:= UNLOCK;

END_ACTION

ACTION FormatDeviceDataProvider:

	// Select CF device if USB device is not available
	FOR i := 0 TO ((SIZEOF(gUSBAvailable) / SIZEOF(gUSBAvailable[0])) - 1) DO
		IF gUSBAvailable[i] THEN
			HmiRecipe.Status.DeviceDataProvider[i + 1] := '{"value":"USB';
			brsitoa(i + 1, ADR(HmiRecipe.Status.DeviceDataProvider[i + 1]) + brsstrlen(ADR(HmiRecipe.Status.DeviceDataProvider[i + 1])));
			brsstrcat(ADR(HmiRecipe.Status.DeviceDataProvider[i + 1]), ADR('","text":"USB'));
			brsitoa(i + 1, ADR(HmiRecipe.Status.DeviceDataProvider[i + 1]) + brsstrlen(ADR(HmiRecipe.Status.DeviceDataProvider[i + 1])));
			brsstrcat(ADR(HmiRecipe.Status.DeviceDataProvider[i + 1]), ADR('"}'));
			MpFileManagerUIConnect.DeviceList.DeviceNames[i + 1] := 'USB';
			brsitoa(i + 1, ADR(MpFileManagerUIConnect.DeviceList.DeviceNames[i + 1]) + brsstrlen(ADR(MpFileManagerUIConnect.DeviceList.DeviceNames[i + 1])));
		ELSE
			brsmemset(ADR(HmiRecipe.Status.DeviceDataProvider[i + 1]), 0, SIZEOF(HmiRecipe.Status.DeviceDataProvider[i + 1]));
			brsmemset(ADR(MpFileManagerUIConnect.DeviceList.DeviceNames[i + 1]), 0, SIZEOF(MpFileManagerUIConnect.DeviceList.DeviceNames[i + 1]));
		END_IF
	END_FOR

END_ACTION

ACTION LoadStatus:
	// Configure recipe actions
	HmiRecipe.Status.FilesAvailable := (MpRecipeUIConnect.Recipe.List.Names[0] <> '');
	HmiRecipe.Status.LoadAllowed := HmiRecipe.Status.FilesAvailable AND NOT HmiRecipe.Status.InvalidRecipe;
	HmiRecipe.Status.DeviceValid := (MpFileManagerUIRecipe.StatusID <> mpFILE_ERR_INVALID_FILE_DEV);

END_ACTION

ACTION LoadPreview:

	//Invalid Recip Manager
	IF HmiRecipe.Status.InvalidRecipe THEN
		HmiRecipe.Status.InvalidRecipeLayer := USINT_TO_BOOL(DISPLAY);
	ELSE
		HmiRecipe.Status.InvalidRecipeLayer := USINT_TO_BOOL(HIDE);
	END_IF;

	// Category name genarate
	IF HmiRecipe.Parameters.CategoryIndex = PARAMETERS_CATEGORY_INDEX THEN
		MpRecipeUIConnect.Recipe.Filter := '*par';
		HmiRecipe.Parameters.Category := PARAMETERS_CATEGORY;
	ELSIF HmiRecipe.Parameters.CategoryIndex = MACH_CONFIG_CATEGORY_INDEX THEN
		MpRecipeUIConnect.Recipe.Filter := '*mcfg';
		HmiRecipe.Parameters.Category := MACHINE_CONFIGURATION_CATEGORY;
	END_IF;
	IF EDGEPOS(HmiRecipe.Parameters.CategoryIndex = PARAMETERS_CATEGORY_INDEX) OR
		EDGEPOS(HmiRecipe.Parameters.CategoryIndex = MACH_CONFIG_CATEGORY_INDEX) THEN
		MpRecipeUIConnect.Recipe.Refresh := TRUE;
	END_IF;

	// Default recipe create Layer manager
	IF HmiRecipe.Status.CreateRecipeLayer.ParsStatus = HIDE AND HmiRecipe.Status.CreateRecipeLayer.MachConfigStatus = HIDE AND
		((HmiRecipe.Status.ParameterRecipeMissing AND HmiRecipe.Parameters.Category = PARAMETERS_CATEGORY) OR
		(HmiRecipe.Status.MachineSettingsRecipeMissing AND HmiRecipe.Parameters.Category = MACHINE_CONFIGURATION_CATEGORY)) THEN
		HmiRecipe.Status.DefaultRecipeLayer.Status := DISPLAY;
	ELSE
		HmiRecipe.Status.DefaultRecipeLayer.Status := HIDE;
	END_IF;

	// Create Recipe Layer manager
	IF HmiRecipe.Parameters.Category = PARAMETERS_CATEGORY THEN
		IF HmiRecipe.Status.CreateDialogOpened THEN
			HmiRecipe.Status.CreateRecipeLayer.ParsStatus := DISPLAY;
		END_IF;
		IF HmiRecipe.Status.CreateRecipeLayer.ParsStatus = DISPLAY AND
			(MpRecipeUIConnect.MessageBox.Cancel OR HmiRecipe.Commands.CreateRecipe) THEN
			HmiRecipe.Status.CreateRecipeLayer.ParsStatus := HIDE;
		END_IF;

	ELSIF HmiRecipe.Parameters.Category = MACHINE_CONFIGURATION_CATEGORY THEN
		IF HmiRecipe.Status.CreateDialogOpened THEN
			HmiRecipe.Status.CreateRecipeLayer.MachConfigStatus := DISPLAY;
		END_IF;
		IF HmiRecipe.Status.CreateRecipeLayer.MachConfigStatus = DISPLAY AND
			(MpRecipeUIConnect.MessageBox.Cancel OR HmiRecipe.Commands.CreateRecipe) THEN
			HmiRecipe.Status.CreateRecipeLayer.MachConfigStatus := HIDE;
		END_IF;
	END_IF;

	// Lock File name input in create layer
	IF HmiRecipe.Status.CreateRecipeLayer.ParsStatus = DISPLAY AND
		HmiRecipe.Status.ParameterRecipeMissing THEN
		HmiRecipe.Status.CreateRecipeLayer.FileNameInputActive	:= LOCK;
	ELSIF HmiRecipe.Status.CreateRecipeLayer.MachConfigStatus = DISPLAY AND
		HmiRecipe.Status.MachineSettingsRecipeMissing THEN
		HmiRecipe.Status.CreateRecipeLayer.FileNameInputActive	:= LOCK;
	ELSE
		HmiRecipe.Status.CreateRecipeLayer.FileNameInputActive	:= UNLOCK;
	END_IF;

	// File Duplicate manager
	IF HmiRecipe.Commands.CreateRecipe AND
		HmiRecipe.Status.FileDuplicate AND
		HmiRecipe.Status.DuplicateLayer = HIDE THEN

		HmiRecipe.Commands.CreateRecipe := FALSE;
		HmiRecipe.Status.DuplicateLayer := DISPLAY;

	ELSIF HmiRecipe.Commands.CreateRecipe THEN
		HmiRecipe.Status.DuplicateLayer := HIDE;
	END_IF;

	// Preview Recipe Layer manager
	IF HmiRecipe.Parameters.Category = MACHINE_CONFIGURATION_CATEGORY THEN
		HmiRecipe.Status.PreviewRecipeLayer.ParsStatus		 := HIDE;
		HmiRecipe.Status.PreviewRecipeLayer.MachConfigStatus := DISPLAY;

	ELSIF HmiRecipe.Parameters.Category = PARAMETERS_CATEGORY THEN
		HmiRecipe.Status.PreviewRecipeLayer.MachConfigStatus := HIDE;
		HmiRecipe.Status.PreviewRecipeLayer.ParsStatus		 := DISPLAY;
	END_IF;

	// Active Recipe declare
	IF HmiRecipe.Parameters.Category = PARAMETERS_CATEGORY THEN
		HmiRecipe.Status.ActiveRecipe := HmiRecipe.Status.LastLoadedProductRecipe;

	ELSIF HmiRecipe.Parameters.Category = MACHINE_CONFIGURATION_CATEGORY THEN
		HmiRecipe.Status.ActiveRecipe := HmiRecipe.Status.LastLoadedConfigRecipe;
	END_IF;

	// Recipe Edit manager
	IF HmiRecipe.Status.EditRecipeLayer.Save THEN
		HmiRecipe.Status.EditRecipeLayer.Save			  := FALSE;
		HmiRecipe.Status.EditRecipeLayer.ParsStatus		  := HIDE;
		HmiRecipe.Status.EditRecipeLayer.MachConfigStatus := HIDE;

		HmiRecipe.Commands.SaveSelectedRecipe := TRUE;
	END_IF;

	// Load preview when a recipe is selected
	IF ((MpRecipeUIConnect.Recipe.List.SelectedIndex <> HmiRecipe.Status.LastSelectedIndex) OR
		(HmiRecipe.Status.LastMaxSelection <> MpRecipeUIConnect.Recipe.List.MaxSelection) OR
		EDGENEG(HmiRecipe.Status.LastStatus = mpRECIPE_UI_STATUS_CREATE)) AND NOT MpRecipeUIConnect.Recipe.Load THEN
		// Check selected recipe name is not empty
		IF (brsstrlen(ADR(MpRecipeUIConnect.Recipe.List.Names[MpRecipeUIConnect.Recipe.List.SelectedIndex])) > 0) THEN
			MpRecipeSys.FileName := ADR(MpRecipeUIConnect.Recipe.List.Names[MpRecipeUIConnect.Recipe.List.SelectedIndex]);
			MpRecipeSys.Category := ADR(HmiRecipe.Parameters.Category);
			MpRecipeSys.Load := TRUE;
			HmiRecipe.Status.LastSelectedIndex := MpRecipeUIConnect.Recipe.List.SelectedIndex;
			HmiRecipe.Status.LastMaxSelection := MpRecipeUIConnect.Recipe.List.MaxSelection;
			HmiRecipe.Status.InvalidRecipe := FALSE;
		END_IF
	END_IF

	// Reset load command on MpRecipeSys FUB
	IF MpRecipeSys.StatusID <> 0 THEN
		HmiRecipe.Status.InvalidRecipe := TRUE;
		HmiRecipe.Commands.ResetPreview := TRUE;
	END_IF;

	IF ((MpRecipeSys.CommandDone) OR (MpRecipeSys.Error)) THEN
		MpRecipeSys.Load := FALSE;
	END_IF

END_ACTION

ACTION RecipeHMIcommands:

	CASE HmiRecipe.Status.HMIcommand OF
		REC_HMI_WAIT:
			// The following commands are triggered directly from the HMI. If you imported the mapp View front end of
			// the Framework, then this is already taken care of. If you did not, then your visualization must
			// trigger each one of these command variables (CreateRecipe, SaveSelectedRecipe, LoadRecipe).
			IF (MpRecipeUIConnect.Status <> mpRECIPE_UI_STATUS_IDLE) THEN
				// MpRecipe is active so don't issue a new command
			ELSIF HmiRecipe.Commands.CreateRecipe THEN
				HmiRecipe.Status.HMIcommand := REC_HMI_CREATE;
				HmiRecipe.Commands.CreateRecipe := FALSE;
			ELSIF HmiRecipe.Commands.SaveSelectedRecipe THEN
				HmiRecipe.Status.HMIcommand := REC_HMI_SAVE;
				HmiRecipe.Commands.SaveSelectedRecipe := FALSE;
			ELSIF HmiRecipe.Commands.LoadRecipe THEN
				HmiRecipe.Status.HMIcommand := REC_HMI_LOAD;
				HmiRecipe.Status.RecipeLoadLayer.Status := HIDE;
				HmiRecipe.Commands.LoadRecipe := FALSE;
				IF (brsstrcmp(ADR(HmiRecipe.Parameters.Category), ADR(PARAMETERS_RECIPE)) = 0) THEN
					HmiRecipe.Status.ProductRecipeLoaded := FALSE;
				ELSE
					HmiRecipe.Status.ConfigRecipeLoaded := FALSE;
				END_IF
			ELSIF HmiRecipe.Commands.ResetPreview THEN
				HmiRecipe.Status.HMIcommand := REC_HMI_RESET_PREVIEW;
				HmiRecipe.Commands.ResetPreview := FALSE;
			END_IF

		REC_HMI_CREATE:
			IF (brsstrcmp(ADR(HmiRecipe.Parameters.Category), ADR(PARAMETERS_RECIPE)) = 0) THEN
				ParametersPreview := ParametersEdit;
				brsstrcpy(ADR(MpRecipeUIConnect.New.FileName), ADR(HmiRecipe.Parameters.FileName));
				brsstrcat(ADR(MpRecipeUIConnect.New.FileName), ADR('.par'));
				// If the default recipe was initially missing and just now created, immediately load it
				IF HmiRecipe.Status.ParameterRecipeMissing THEN
					HmiRecipe.Commands.LoadRecipe := TRUE;
				END_IF
			ELSIF (brsstrcmp(ADR(HmiRecipe.Parameters.Category), ADR(MACHINE_CONFIGURATION_RECIPE)) = 0) THEN
				MachineSettingsPreview := MachineSettingsEdit;
				brsstrcpy(ADR(MpRecipeUIConnect.New.FileName), ADR(HmiRecipe.Parameters.FileName));
				brsstrcat(ADR(MpRecipeUIConnect.New.FileName), ADR('.mcfg'));
				// If the default recipe was initially missing and just now created, immediately load it
				IF HmiRecipe.Status.MachineSettingsRecipeMissing THEN
					HmiRecipe.Commands.LoadRecipe := TRUE;
				END_IF
			END_IF

			Header.Name := MpRecipeUIConnect.New.FileName;
			DTGetTimeRecipe.enable := TRUE;
			REPEAT
				DTGetTimeRecipe();
				UNTIL (DTGetTimeRecipe.status = 0)
			END_REPEAT;
			Header.DateTime := DTGetTimeRecipe.DT1;
			DTGetTimeRecipe.enable := FALSE;
			DTGetTimeRecipe();
			MpRecipeUIConnect.New.Create := TRUE;

			HmiRecipe.Status.HMIcommand := REC_HMI_WAIT;

		REC_HMI_LOAD:
			IF (MpRecipeUIConnect.Status = mpRECIPE_UI_STATUS_IDLE) THEN
				IF (brsstrcmp(ADR(HmiRecipe.Parameters.Category), ADR(PARAMETERS_RECIPE)) = 0) THEN
					Parameters := ParametersPreview;
					HmiRecipe.Status.ProductRecipeLoaded := TRUE;
					// If the default recipe was initially missing and just now created, then it is the last loaded recipe
					IF HmiRecipe.Status.ParameterRecipeMissing THEN
						HmiRecipe.Status.LastLoadedProductRecipe := DEFAULT_PARAMETERS;
						brsstrcat(ADR(HmiRecipe.Status.LastLoadedProductRecipe), ADR(PARAMETERS_FILE_EXTENSION));
						HmiRecipe.Status.ParameterRecipeMissing := FALSE;
						// Otherwise, the last loaded recipe is the selected recipe
					ELSE
						HmiRecipe.Status.LastLoadedProductRecipe := MpRecipeUIConnect.Recipe.List.Names[MpRecipeUIConnect.Recipe.List.SelectedIndex];
					END_IF
				ELSIF (brsstrcmp(ADR(HmiRecipe.Parameters.Category), ADR(MACHINE_CONFIGURATION_RECIPE)) = 0) THEN
					MachineSettings := MachineSettingsPreview;
					HmiRecipe.Status.ConfigRecipeLoaded := TRUE;
					// If the default recipe was initially missing and just now created, then it is the last loaded recipe
					IF HmiRecipe.Status.MachineSettingsRecipeMissing THEN
						HmiRecipe.Status.LastLoadedConfigRecipe := DEFAULT_MACHINE_CONFIGURATION;
						brsstrcat(ADR(HmiRecipe.Status.LastLoadedConfigRecipe), ADR(MACHINE_CONFIG_FILE_EXTENSION));
						HmiRecipe.Status.MachineSettingsRecipeMissing := FALSE;
						// Otherwise, the last loaded recipe is the selected recipe
					ELSE
						HmiRecipe.Status.LastLoadedConfigRecipe := MpRecipeUIConnect.Recipe.List.Names[MpRecipeUIConnect.Recipe.List.SelectedIndex];
					END_IF
				END_IF
				HmiRecipe.Status.HMIcommand := REC_HMI_WAIT;
			END_IF

		REC_HMI_SAVE:
			IF (MpRecipeUIConnect.Status = mpRECIPE_UI_STATUS_IDLE) THEN

				IF (brsstrcmp(ADR(HmiRecipe.Parameters.Category), ADR(PARAMETERS_RECIPE)) = 0) THEN
					ParametersPreview := ParametersEdit;
				ELSIF (brsstrcmp(ADR(HmiRecipe.Parameters.Category), ADR(MACHINE_CONFIGURATION_RECIPE)) = 0) THEN
					MachineSettingsPreview := MachineSettingsEdit;
				END_IF

				IF (brsstrlen(ADR(HmiRecipe.Status.SelectedRecipe)) > 0) THEN
					MpRecipeSys.FileName := ADR(HmiRecipe.Status.SelectedRecipe);
					MpRecipeSys.Save := TRUE;
				END_IF

				HmiRecipe.Status.HMIcommand := REC_HMI_WAIT;
			END_IF

		REC_HMI_RESET_PREVIEW:
			IF (brsstrcmp(ADR(HmiRecipe.Parameters.Category), ADR(PARAMETERS_RECIPE)) = 0) THEN
				brsmemset(ADR(ParametersPreview), 0, SIZEOF(ParametersPreview));
			ELSIF (brsstrcmp(ADR(HmiRecipe.Parameters.Category), ADR(MACHINE_CONFIGURATION_RECIPE)) = 0) THEN
				brsmemset(ADR(MachineSettingsPreview), 0, SIZEOF(MachineSettingsPreview));
			END_IF
			HmiRecipe.Status.HMIcommand := REC_HMI_WAIT;

	END_CASE

	//default files cannot be deleted
	IF HmiRecipe.Status.SelectedRecipe = 'Default.par' OR
		HmiRecipe.Status.SelectedRecipe = 'Machine.mcfg' THEN

		HmiRecipe.Status.DefaultFilesDeleteButtonStatus := DISPLAY;
	ELSE
		HmiRecipe.Status.DefaultFilesDeleteButtonStatus := HIDE;
	END_IF;

	//selected index should be equal active recipe
	IF HmiRecipe.Status.RecipePageOpenedNow THEN
		HmiRecipe.Status.LoadPreviewAfterPageOpened := TRUE;
	END_IF;
	IF EDGEPOS(MpRecipeUIConnect.Status = mpRECIPE_UI_STATUS_IDLE) THEN
		IF HmiRecipe.Status.RecipePageOpenedNow THEN
			HmiRecipe.Status.RecipePageOpenedNow := FALSE;
			FOR i := 0 TO 19 DO
				IF MpRecipeUIConnect.Recipe.List.Names[i] = HmiRecipe.Status.ActiveRecipe THEN
					MpRecipeUIConnect.Recipe.List.SelectedIndex := i;
				END_IF;
			END_FOR;
		END_IF;
	END_IF;
	IF HmiRecipe.Status.LoadPreviewAfterPageOpened THEN
		HmiRecipe.Status.LoadPreviewAfterPageOpened := FALSE;
		// Check selected recipe name is not empty
		IF (brsstrlen(ADR(MpRecipeUIConnect.Recipe.List.Names[MpRecipeUIConnect.Recipe.List.SelectedIndex])) > 0) THEN
			MpRecipeSys.FileName := ADR(MpRecipeUIConnect.Recipe.List.Names[MpRecipeUIConnect.Recipe.List.SelectedIndex]);
			MpRecipeSys.Category := ADR(HmiRecipe.Parameters.Category);
			MpRecipeSys.Load := TRUE;
			HmiRecipe.Status.LastSelectedIndex := MpRecipeUIConnect.Recipe.List.SelectedIndex;
			HmiRecipe.Status.LastMaxSelection := MpRecipeUIConnect.Recipe.List.MaxSelection;
			HmiRecipe.Status.InvalidRecipe := FALSE;
		END_IF
	END_IF;

	// If the Edit or Create dialog boxes open, copy the Preview structure into the Edit structure.
	IF HmiRecipe.Status.EditDialogOpened OR HmiRecipe.Status.CreateDialogOpened THEN
		IF (brsstrcmp(ADR(HmiRecipe.Parameters.Category), ADR(PARAMETERS_RECIPE)) = 0) THEN
			ParametersEdit := ParametersPreview;
			IF HmiRecipe.Status.ParameterRecipeMissing THEN
				HmiRecipe.Parameters.FileName := DEFAULT_PARAMETERS;
			ELSE
				HmiRecipe.Parameters.FileName:= 'newParameters';
			END_IF

			// Open parameter dialog
			IF HmiRecipe.Status.EditDialogOpened THEN
				HmiRecipe.Status.EditRecipeLayer.ParsStatus := DISPLAY;
			ELSIF HmiRecipe.Status.CreateDialogOpened THEN
			END_IF;

		ELSIF (brsstrcmp(ADR(HmiRecipe.Parameters.Category), ADR(MACHINE_CONFIGURATION_RECIPE)) = 0) THEN
			MachineSettingsEdit := MachineSettingsPreview;
			IF HmiRecipe.Status.MachineSettingsRecipeMissing THEN
				HmiRecipe.Parameters.FileName := DEFAULT_MACHINE_CONFIGURATION;
			ELSE
				HmiRecipe.Parameters.FileName := 'newMachineConfig';
			END_IF

			// Open machine dialog
			IF HmiRecipe.Status.EditDialogOpened THEN
				HmiRecipe.Status.EditRecipeLayer.MachConfigStatus := DISPLAY;
			ELSIF HmiRecipe.Status.CreateDialogOpened THEN
			END_IF;

		END_IF

		HmiRecipe.Status.EditDialogOpened := FALSE;
		HmiRecipe.Status.CreateDialogOpened := FALSE;
	END_IF

	// Check if the file name has already been used
	HmiRecipe.Status.FileDuplicate := FALSE;
	FOR i:=0 TO ((SIZEOF(MpRecipeUIConnect.Recipe.List.Names) / SIZEOF(MpRecipeUIConnect.Recipe.List.Names[0])) - 1) DO
		temp := HmiRecipe.Parameters.FileName;
		IF (brsstrcmp(ADR(HmiRecipe.Parameters.Category), ADR(PARAMETERS_RECIPE)) = 0) THEN
			brsstrcat(ADR(temp),ADR(PARAMETERS_FILE_EXTENSION));
		ELSIF (brsstrcmp(ADR(HmiRecipe.Parameters.Category), ADR(MACHINE_CONFIGURATION_RECIPE)) = 0) THEN
			brsstrcat(ADR(temp),ADR(MACHINE_CONFIG_FILE_EXTENSION));
		END_IF
		IF temp = MpRecipeUIConnect.Recipe.List.Names[i] THEN
			HmiRecipe.Status.FileDuplicate := TRUE;
		END_IF
	END_FOR

	// Set whether the loading .gif should be shown on the HMI
	HmiRecipe.Status.LoadingRecipeList := (MpRecipeUIConnect.Status = mpRECIPE_UI_STATUS_REFRESH);

	// Update status information
	HmiRecipe.Status.LastStatus := MpRecipeUIConnect.Status;
	HmiRecipe.Status.SelectedRecipe := MpRecipeUIConnect.Recipe.List.Names[MpRecipeUIConnect.Recipe.List.SelectedIndex];

END_ACTION
```

### Package Logical/Infrastructure/VC4/UserX - Package for mapp UserX Framework

### Program Logical/Infrastructure/VC4/UserX/UserXMgr (IEC)

#### UserXMgr.st - Init, cyclic, exit code
```iecst
//***********************************************************************
// Copyright: B&R Industrial Automation GmbH
// Author: B&R Industrial Automation GmbH
// Created: April 12, 2022
// Description: Tasks for user management with VC4 front-end.
//***********************************************************************

PROGRAM _INIT

	// Create folder for this component on the user file device
	DirCreateUser(enable := TRUE, pDevice := ADR('mappUserXFiles'), pName := ADR('/'));

	// Check if folder already exist and if so disabled the function block call
	IF DirCreateUser.status = fiERR_DIR_ALREADY_EXIST THEN
		DirCreateUser(enable := FALSE);
	END_IF

	 // Initial visibility setup
	VC4_Init;

	// Initialize mapp function blocks
	UserXMgrUIConnect.User.Create.Lock := FALSE;
	UserXMgrUIConnect.User.Lock := FALSE;
	UserXMgrUIConnect.User.Edit.Lock := FALSE;
	UserXMgrUIConnect.User.Create.Dialog.UserName := "";
	UserXMgrUIConnect.User.Create.Dialog.NewPassword := "";
	UserXMgrUIConnect.User.Create.Dialog.ConfirmPassword := "";
	UserXMgrUIConnect.User.List.MaxSelection := USER_LIST_MAX_SELECTION;
	UserXMgrUIConnect.User.List.RangeStart := USER_LIST_RANGE_START;
	UserXMgrUIConnect.User.List.RangeEnd := USER_LIST_RANGE_END;
	MpUserXManagerUISys.MpLink := ADR(gMpLinkUserXLogin);
	MpUserXManagerUISys.Enable := TRUE;
	MpUserXManagerUISys.UIConnect := ADR(UserXMgrUIConnect);
	MpUserXManagerUISys();

	MpUserXLoginUISys.MpLink := ADR(gMpLinkUserXLogin);
	MpUserXLoginUISys.Enable := TRUE;
	MpUserXLoginUISys.UIConnect := ADR(UserXLoginUIConnect);
	MpUserXLoginUISys();

	MpUserXLoginSys.MpLink := ADR(gMpLinkUserXLogin);
	MpUserXLoginSys.Enable := TRUE;
	MpUserXLoginSys();

END_PROGRAM

PROGRAM _CYCLIC

	// Error reset
	IF NOT MpUserXManagerUISys.Error THEN
		MpUserXManagerUISys.ErrorReset := FALSE;
	END_IF

	IF NOT MpUserXLoginUISys.Error THEN
		MpUserXLoginUISys.ErrorReset := FALSE;
	END_IF

	IF NOT MpUserXLoginSys.Error THEN
		MpUserXLoginSys.ErrorReset := FALSE;
	END_IF

	// Cyclic action calls
	VC4_Cylic;

	// Assign MpLinks
	MpUserXManagerUISys.MpLink := ADR(gMpLinkUserXLogin);
	MpUserXManagerUISys.UIConnect := ADR(UserXMgrUIConnect);
	MpUserXLoginUISys.MpLink := ADR(gMpLinkUserXLogin);
	MpUserXLoginUISys.UIConnect := ADR(UserXLoginUIConnect);
	MpUserXLoginSys.MpLink := ADR(gMpLinkUserXLogin);

	// Call function blocks
	MpUserXManagerUISys();
	MpUserXLoginUISys();
	MpUserXLoginSys();

END_PROGRAM

PROGRAM _EXIT

	// Disable the function blocls to unlink the MpLinks
	MpUserXManagerUISys.Enable := FALSE;
	MpUserXLoginUISys.Enable := FALSE;
	MpUserXLoginSys.Enable := FALSE;

	// Call function blocks
	MpUserXManagerUISys();
	MpUserXLoginUISys();
	MpUserXLoginSys();

END_PROGRAM
```

#### UserXMgr.typ - Local data types
```iecst
(*Structure types*)

TYPE
	UserXHmiInterfaceType : 	STRUCT
		NewFileName : STRING[255];
		Export : BOOL;
		ConfirmOverwrite : BOOL;
		CancelOverwrite : BOOL;
		FileDuplicate : BOOL;
		FileDuplicateLayerStatus : USINT;
		ButtonLockedMessageLayer : USINT;
		ButtonLockingLayer : USINT;
		SelectedLanguage : USINT;
		PreviousUser : WSTRING[50];
	END_STRUCT;
END_TYPE

(*Enumerations*)

TYPE
	HmiStateEnum :
		(
		USERX_START := 0,
		USERX_WAIT_FOR_DIALOG := 1,
		USERX_SET_RESPONSE := 2,
		USERX_CONFIRM_RESPONSE := 3,
		USERX_NEW_EXPORT := 4,
		USERX_FINISH := 5
		);
END_TYPE
```

#### UserXMgr.var - Local variables
```iecst
(*Function Blocks*)
VAR
	MpUserXLogin_0 : MpUserXLogin; (*MpUserXLogin instance*)
	MpUserXManagerUI_0 : MpUserXManagerUI := (UISetup:=(FileDevice:='mappUserXFiles')); (*MpUserXManagerUI instance*)
	MpUserXLoginUI_0 : MpUserXLoginUI; (*MpUserXLoginUI instance*)
	DirCreate_0 : DirCreate; (*DirCreate instance*)
END_VAR
(*Constants*)
VAR CONSTANT
	DISPLAY : USINT := 0;
	HIDE : USINT := 1;
	USER_ADMIN_LEVEL : USINT := 100;
END_VAR
(**)
VAR CONSTANT
	USER_LIST_MAX_SELECTION : USINT := 20; (*Maxiumum selections on the User List *)
	USER_LIST_RANGE_START : USINT := 0; (*Range start (used for UserXMgrUIConnect)*)
	USER_LIST_RANGE_END : USINT := 20; (*Range end (used for UserXMgrUIConnect)*)
END_VAR
(*Structure Types*)
VAR
	UserXMgrUIConnect : MpUserXMgrUIConnectType; (*UserX manager connection to the HMI*)
	UserXLoginUIConnect : MpUserXLoginUIConnectType; (*UserL login connection to the HMI*)
	i : USINT;
	HmiUserX : HMIUser_Typ;
END_VAR
(*Enumerations*)
(*Variables*)
VAR
	UserXCheckState : enumCheckState;
	temp : STRING[255]; (*Temporary string holder for checking file names*)
END_VAR
```

#### HMIAction.st
```iecst
ACTION VC4_Init:

	HmiUserX.FileDuplicateLayerStatus := HIDE;
	HmiUserX.ButtonLockedMessageLayer := HIDE;
	UserXLoginUIConnect.ChangePassword.Dialog.LayerStatus := HIDE;

END_ACTION

ACTION VC4_Cylic:

	CASE UserXCheckState OF
		USERX_START:
			IF NOT UserXMgrUIConnect.Import.ShowDialog THEN
				UserXMgrUIConnect.Import.ShowDialog := TRUE;
			ELSE
				UserXCheckState := USERX_WAIT_FOR_DIALOG;
			END_IF
		USERX_WAIT_FOR_DIALOG:
			UserXMgrUIConnect.Import.ShowDialog := FALSE;
			UserXCheckState := USERX_SET_RESPONSE;
		USERX_SET_RESPONSE:
			IF NOT(UserXMgrUIConnect.Status = mpUSERX_UI_STATUS_IDLE) THEN
				UserXMgrUIConnect.Import.Dialog.Cancel := TRUE;
			ELSE
				UserXMgrUIConnect.Import.Dialog.Cancel := FALSE;
				UserXCheckState := USERX_CONFIRM_RESPONSE;
			END_IF
		USERX_CONFIRM_RESPONSE:
			IF UserXMgrUIConnect.Status = mpUSERX_UI_STATUS_WAIT_DLG THEN
				UserXCheckState := USERX_START;
			ELSE
				UserXCheckState := USERX_FINISH;
			END_IF
		USERX_NEW_EXPORT:
			IF NOT UserXMgrUIConnect.Export.ShowDialog AND UserXMgrUIConnect.Status = mpUSERX_UI_STATUS_IDLE THEN
				UserXCheckState := USERX_START;
			END_IF
		USERX_FINISH:

	END_CASE

	// Assign file name based on selected index
	UserXMgrUIConnect.Import.Dialog.FileName := UserXMgrUIConnect.Import.Dialog.List.FileNames[UserXMgrUIConnect.Import.Dialog.List.SelectedIndex];

	// If new updates are made via export execute a check
	IF UserXMgrUIConnect.Export.ShowDialog THEN
		UserXCheckState := USERX_NEW_EXPORT;
	END_IF

	// Check User is Admin
	IF UserXLoginUIConnect.UserLevel = USER_ADMIN_LEVEL THEN
		HmiUserX.ButtonLockingLayer := HIDE;
	ELSE
		HmiUserX.ButtonLockingLayer := DISPLAY;
	END_IF;

	// Duplicate file checks
	HmiUserX.FileDuplicate := FALSE;
	FOR i := 0 TO ((SIZEOF(UserXMgrUIConnect.Import.Dialog.List.FileNames) / SIZEOF(UserXMgrUIConnect.Import.Dialog.List.FileNames[0])) - 1) DO
		temp := UserXMgrUIConnect.Export.Dialog.FileName;
		brsstrcat(ADR(temp),ADR('.usr'));
		IF (temp = UserXMgrUIConnect.Import.Dialog.List.FileNames[i]) AND HmiUserX.Export THEN
			HmiUserX.FileDuplicate := TRUE;
		END_IF
	END_FOR

	IF HmiUserX.FileDuplicate AND (HmiUserX.ConfirmOverwrite) THEN
		UserXMgrUIConnect.Export.Dialog.Confirm := TRUE;
		HmiUserX.Export := FALSE;
		HmiUserX.FileDuplicate := FALSE;

	ELSIF HmiUserX.FileDuplicate AND (HmiUserX.CancelOverwrite) THEN
		UserXMgrUIConnect.Export.Dialog.Cancel := TRUE;
		HmiUserX.Export := FALSE;
		HmiUserX.FileDuplicate := FALSE;

	ELSIF NOT HmiUserX.FileDuplicate AND HmiUserX.Export THEN
		UserXMgrUIConnect.Export.Dialog.Confirm := TRUE;
		HmiUserX.Export := FALSE;

	ELSIF NOT HmiUserX.FileDuplicate AND UserXMgrUIConnect.Export.Dialog.Cancel THEN
		UserXMgrUIConnect.Export.Dialog.Cancel := TRUE;
		HmiUserX.Export := FALSE;
	END_IF

	// Manage FileExport Layer - close
	IF UserXMgrUIConnect.Export.Dialog.Cancel OR HmiUserX.Export THEN
		UserXMgrUIConnect.Export.Dialog.LayerStatus := HIDE;
	END_IF

	// Manage FileDupliacte Layer - close
	IF HmiUserX.CancelOverwrite OR HmiUserX.ConfirmOverwrite THEN
		HmiUserX.CancelOverwrite := FALSE;
		HmiUserX.ConfirmOverwrite := FALSE;
		HmiUserX.FileDuplicateLayerStatus := HIDE;
	END_IF

	// Manage FileDupliacte Layer - open
	IF HmiUserX.Export AND HmiUserX.FileDuplicate THEN
		HmiUserX.FileDuplicateLayerStatus := DISPLAY;
	END_IF;

	// Password change require manage
	IF EDGENEG(UserXLoginUIConnect.MessageBox.ErrorNumber = 28690) THEN
		IF UserXLoginUIConnect.MessageBox.Confirm THEN
			UserXLoginUIConnect.ChangePassword.Dialog.LayerStatus := DISPLAY;
			UserXLoginUIConnect.ChangePassword.ShowDialog := TRUE;
		END_IF
	END_IF

	// Check and set current language datapoint based on user preference
	IF UserXLoginUIConnect.CurrentUser <> HmiUserX.PreviousUser THEN
		HmiUserX.PreviousUser := UserXLoginUIConnect.CurrentUser;
		IF UserXLoginUIConnect.Language = 'en' THEN
			HmiUserX.SelectedLanguage := 0;
		ELSIF UserXLoginUIConnect.Language = 'de' THEN
			HmiUserX.SelectedLanguage := 1;
		ELSIF UserXLoginUIConnect.Language = 'zh' THEN
			HmiUserX.SelectedLanguage := 2;
		END_IF
	END_IF

END_ACTION
```

### Package Logical/Infrastructure/VC4/Audit - Package for mapp Audit Framework

### Program Logical/Infrastructure/VC4/Audit/AuditMgr (IEC) - Audit manager

#### AuditMgr.typ
```iecst
TYPE
	AuditQueryHMIType : 	STRUCT  (*Datatype for the structure which rearranges the query data from AuditQuery into a structure of arrays for easy connection to the Table widget in mapp View*)
		EvTime : ARRAY[0..MAX_QUERY_RESULTS]OF DATE_AND_TIME; (*ActiveAudits query, Event-Time column*)
		EvTimeString : ARRAY[0..MAX_QUERY_RESULTS]OF STRING[80]; (*ActiveAudits query, Event-Time column*)
		Text : ARRAY[0..MAX_QUERY_RESULTS]OF WSTRING[100]; (*ActiveAudits query, Text column*)
		DText : ARRAY[0..MAX_QUERY_RESULTS]OF WSTRING[100]; (*ActiveAudits query, Display Text column*)
		Op : ARRAY[0..MAX_QUERY_RESULTS]OF WSTRING[100]; (*ActiveAudits query, Operator-Name column*)
		QueryCount : USINT; (*Count of query results for building the query table configuration string*)
		Name : STRING[80]; (*Name of the query to be executed*)
		Option : USINT; (*Index value of the selected query type in the dropdown on the query tab*)
		DPSelectedIndex : USINT;
	END_STRUCT;
	ActiveAuditStateEnum :
		( (*Enumeration for the state for the query state machine*)
		ACTIVE_AUDIT_WAIT, (*Wait state*)
		ACTIVE_AUDIT_QUERY, (*State to query the Audit data*)
		ACTIVE_AUDIT_NEXT (*State to check if more Audits meet the query criteria and need to be queried*)
		);
	AuditCustomEventType : 	STRUCT  (*Structure for custom events handling*)
		Set : BOOL; (*Trigger the assigned function*)
		Type : WSTRING[100]; (*Entered when creating the entry under %typ*)
		Msg : WSTRING[100]; (*Entered when creating the entry under %msg *)
		Comment : WSTRING[100]; (*Entered when creating the entry under %cmt *)
	END_STRUCT;
	AuditQueryType : 	STRUCT  (*Structure for query results and status*)
		State : ActiveAuditStateEnum; (*State variable for the query state machine*)
		LastUpdateCount : UDINT; (*Previous count of query results. Used to check for new query data. *)
		UpdateCountRecipe : UDINT; (*Count of query results. Increases each time new results are availble. *)
		UpdateCount : UDINT; (*Count of query results. Increases each time new results are availble. *)
		Audits : ARRAY[0..MAX_QUERY_RESULTS]OF AuditType; (*Query data*)
		Next : BOOL; (*Trigger to query the next data, if there are more results than MAX_QUERY_RESULTS*)
	END_STRUCT;
	AuditHmiInterfaceType : 	STRUCT  (*Structure to hold commands and status from the HMI*)
		Commands : AuditCommandsType; (*HMI commands*)
		Parameters : AuditParType; (*HMI parameters*)
		Status : {REDUND_UNREPLICABLE} AuditStatusType; (*HMI status*)
	END_STRUCT;
	AuditCommandsType : 	STRUCT  (*Structure to hold the commands from the HMI*)
		ExportArchives : BOOL; (*Triggers an Audit export of the Audit history. Connected to a button on the HMI. *)
		RunQuery : BOOL; (*Triggers the query to run. Connected to a button on the HMI. *)
		SaveConfig : BOOL; (*Starts the configuration for archives*)
	END_STRUCT;
	AuditStatusType : 	STRUCT  (*Structure to hold status information from the mapp View HMI. (This structure is not compatible/relevant if you are using a VC4 visualization)*)
		AuditSortCfg : STRING[1000]; (*Sort configuration for the AuditList widget*)
		AuditFilterCfg : STRING[1000]; (*Filter configuration for the AuditList widget*)
		TableConfig : ARRAY[0..1]OF STRING[255]; (*Table configuration for the Audit query Table*)
		Query : AuditQueryHMIType; (*Structure which rearranges the query data from AuditQuery into a structure of arrays for easy connection to the Table widget*)
		CustomEventSortCfg : STRING[1000]; (*Sort configuration for the AuditList Custom Events widget*)
		CustomEventsFilterCfg : STRING[1000]; (*Filter configuration for the AuditList Custom Events widget*)
		ArchiveAvailable : BOOL; (*At least 1 archive is available for export*)
		NumberOfArchives : UINT; (*How many archives are available for export*)
		DeviceDataProvider : ARRAY[0..1]OF STRING[100]; (*Data provider for the file device selector*)
		DeviceDataProviderVC4 : ARRAY[0..1]OF STRING[100]; (*Data provider for the file device selector*)
		ArchiveSetupLayer : USINT;
		ArchiveSetupTimeOfDayVisibility : USINT;
		ArchiveSetupVisibility : USINT;
	END_STRUCT;
	AuditParType : 	STRUCT  (*Structure to hold parameter data for the HMI*)
		ArchiveSettings : AuditArchiveParType; (*Parameter for archive configuration*)
		QuerySelection : ARRAY[0..MAX_QUERIES]OF STRING[10]; (*The selection in the query dropdown on the query tab of the Audit content*)
	END_STRUCT;
	AuditArchiveParType : 	STRUCT  (*Automatic archive settings*)
		Enable : BOOL; (*Enable automatic archive feature*)
		MaxSize : UDINT; (*Name prefix for each automatic backup file*)
		Mode : MpAuditArchiveModeEnum; (*Mode (daily, Mo-Fr or by batch)*)
		Hour : USINT; (*Time (hour)*)
		Minute : USINT; (*Time (minutes)*)
		FileType : MpAuditFileTypeEnum := mpAUDIT_FILE_TYPE_XML; (*File type selection (XML, TXT, PDF)*)
	END_STRUCT;
	AuditType : 	STRUCT  (*Structure to hold the Audit data for the query results*)
		EvTime : DATE_AND_TIME; (*ActiveAudits query, Event-Time column*)
		Text : WSTRING[100]; (*ActiveAudits query, Text column*)
		DText : WSTRING[100]; (*ActiveAudits query, Display Text column*)
		Op : WSTRING[100]; (*ActiveAudits query, Operator-Name column*)
	END_STRUCT;
END_TYPE

(*Enumerations*)
```

#### AuditMgr.var
```iecst
(*Function Blocks*)
VAR
	DirCreateAudit : DirCreate; (*DirCreate instance*)
	MpAuditTrailSys : MpAuditTrail; (*AuditTrail for regular mapp events*)
	MpAuditTrailConfigSys : MpAuditTrailConfig; (*AuditTrail configuration*)
	MpAuditTrailCEvents : MpAuditTrail; (*AuditTrail for custom events*)
	QueryUserEvents : {REDUND_UNREPLICABLE} MpAuditQuery; (*MpAlarmXQuery instance*)
	MpAuditTrailUISys : MpAuditTrailUI; (*AuditTrail UI interface*)
	MpAuditTrailCEventsUI : MpAuditTrailUI; (*AuditTrail UI interface*)
END_VAR
(*Constants*)
VAR CONSTANT
	MAX_QUERY_RESULTS : USINT := 19; (*Maximum number of query results (Value+1)*)
	MAX_CUSTOM_EVENTS : USINT := 9; (*Maximum number of custom events*)
	MAX_QUERIES : USINT := 2; (*Maximum number of configured queries*)
END_VAR
(*Structure Types*)
VAR
	HmiAudit : AuditHmiInterfaceType; (*HMI interface structure*)
	CustomEvent : ARRAY[0..MAX_CUSTOM_EVENTS] OF AuditCustomEventType; (*Custom events*)
	AuditQuery : {REDUND_UNREPLICABLE} AuditQueryType; (*Query results and status*)
	AuditTrailConfig : MpAuditTrailConfigType; (*Configuration structure for changing archiving setup*)
	MpAuditTrailUIConnect : MpAuditTrailUIConnectType; (*MpAuditUI connection to the HMI*)
END_VAR
VAR RETAIN
	ArchiveSettingsRetain : AuditArchiveParType; (*Store settings in retain memory to be applied after boot*)
END_VAR
VAR
	MpAuditTrailCEventsUIConnect : MpAuditTrailUIConnectType; (*MpAuditUI connection to the HMI*)
END_VAR
(*Variables*)
VAR
	i : USINT; (*Index for loops*)
	ident : UDINT; (*Identifier for task deployment*)
	VariableMonitorExample : REAL; (*Used for the variable monitor example*)
END_VAR
```

#### AuditMgr.st
```iecst
//***********************************************************************
// Copyright: B&R Industrial Automation GmbH
// Author: B&R Industrial Automation GmbH
// Created: Sept 1, 2022
// Description: Task for audit management with VC4 front-end.
//***********************************************************************

PROGRAM _INIT

	// Create folder for this component on the user file device
	DirCreateAudit(enable := TRUE, pDevice := ADR('mappAuditFiles'), pName := ADR('/'));

	// Check if folder already exist and if so disabled the function block call
	IF DirCreateAudit.status = fiERR_DIR_ALREADY_EXIST THEN
		DirCreateAudit(enable := FALSE);
	END_IF

	// Initialize mapp function blocks
	MpAuditTrailSys.Enable := TRUE;
	MpAuditTrailSys.MpLink := ADR(gMpLinkAuditTrail);
	MpAuditTrailSys.Language := ADR('en');
	MpAuditTrailSys.DeviceName := ADR('mappAuditFiles');
	MpAuditTrailSys();

	MpAuditTrailConfigSys.Enable := TRUE;
	MpAuditTrailConfigSys.MpLink := ADR(gMpLinkAuditTrail);
	MpAuditTrailConfigSys.Configuration := ADR(AuditTrailConfig);
	MpAuditTrailConfigSys.Load := TRUE;
	MpAuditTrailConfigSys();

	MpAuditTrailCEvents.Enable := TRUE;
	MpAuditTrailCEvents.MpLink := ADR(gMpLinkCustomEvents);
	MpAuditTrailCEvents();

	MpAuditTrailUISys.MpLink := ADR(gMpLinkAuditTrail);
	MpAuditTrailUISys.UIConnect := ADR(MpAuditTrailUIConnect);
	MpAuditTrailUISys.UISetup.EventListSize := SIZEOF(MpAuditTrailUIConnect.Output.EventID) / SIZEOF(MpAuditTrailUIConnect.Output.EventID[0]);
	MpAuditTrailUISys.UISetup.ScrollWindow := 1;
	MpAuditTrailUISys.Enable := TRUE;
	MpAuditTrailUISys();

	MpAuditTrailCEventsUI.MpLink := ADR(gMpLinkCustomEvents);
	MpAuditTrailCEventsUI.UIConnect := ADR(MpAuditTrailCEventsUIConnect);
	MpAuditTrailCEventsUI.UISetup.EventListSize := SIZEOF(MpAuditTrailCEventsUIConnect.Output.EventID) / SIZEOF(MpAuditTrailCEventsUIConnect.Output.EventID[0]);
	MpAuditTrailCEventsUI.UISetup.ScrollWindow := 1;
	MpAuditTrailCEventsUI.Enable := TRUE;
	MpAuditTrailCEventsUI();

	// Initialize custom events
	CustomEvent[0].Type := "Custom Event Type";
	CustomEvent[0].Msg := "Custom Event Message";
	CustomEvent[0].Comment := "Custom Event Comment";

	CustomEvent[1].Type := "Audit Test";
	CustomEvent[1].Msg := "This is a custom event test msg";
	CustomEvent[1].Comment := "If you see this it was a success!";

	CustomEvent[2].Type := "Cmd Exe";
	CustomEvent[2].Msg := "The run query command was pressed on the HMI";
	CustomEvent[2].Comment := "Result can be seen in the Query tab";

	HmiAudit.Status.Query.Name := 'UserEvents';
	HmiAudit.Status.Query.Option := 1;

	// Configuring the query selection, reading the available components
	HmiAudit.Parameters.QuerySelection[0] := 'UserXMgr';
	HmiAudit.Parameters.QuerySelection[1] := 'RecipeMgr';

	IF (ST_ident(ADR(HmiAudit.Parameters.QuerySelection[0]), 0, ADR(ident)) = 0) AND (ST_ident(ADR(HmiAudit.Parameters.QuerySelection[1]), 0, ADR(ident)) = 0) THEN
		HmiAudit.Status.DeviceDataProvider[0] := '{"value":"UserEvents","text":"User Events Query"}';
		HmiAudit.Status.DeviceDataProvider[1] := '{"value":"RecipeEvents","text":"Recipe Events Query"}';

		HmiAudit.Status.DeviceDataProviderVC4[0] := 'User Events Query';
		HmiAudit.Status.DeviceDataProviderVC4[1] := 'Recipe Events Query';

	ELSIF (ST_ident(ADR(HmiAudit.Parameters.QuerySelection[0]), 0, ADR(ident)) <> 0) AND (ST_ident(ADR(HmiAudit.Parameters.QuerySelection[1]), 0, ADR(ident)) = 0) THEN
		HmiAudit.Status.DeviceDataProvider[0] := '{"value":"RecipeEvents","text":"Recipe Events Query"}';

		HmiAudit.Status.DeviceDataProviderVC4[0] := 'Recipe Events Query';

	ELSIF (ST_ident(ADR(HmiAudit.Parameters.QuerySelection[0]), 0, ADR(ident)) = 0) AND (ST_ident(ADR(HmiAudit.Parameters.QuerySelection[1]), 0, ADR(ident)) <> 0) THEN
		HmiAudit.Status.DeviceDataProvider[0] := '{"value":"UserEvents","text":"User Events Query"}';

		HmiAudit.Status.DeviceDataProviderVC4[0] := 'User Events Query';
	END_IF

	// Restored the retained values to the archive settings
	HmiAudit.Parameters.ArchiveSettings := ArchiveSettingsRetain;

END_PROGRAM

PROGRAM _CYCLIC

	// Call all cyclic actions
	ExecuteQuery;
	ArchiveExport;
	ArchiveSettings;
	ChangeConfiguration;
	VC4_Cyclic;

	// Sample code for how custom events can be triggered. Use custom events as needed around the application for debugging purposes.
	IF EDGEPOS(CustomEvent[0].Set) THEN
		MpAuditCustomEvent(gMpLinkCustomEvents,CustomEvent[0].Type,CustomEvent[0].Msg,CustomEvent[0].Comment);
	END_IF
	IF EDGENEG(CustomEvent[1].Set) THEN
		MpAuditCustomEvent(gMpLinkCustomEvents,CustomEvent[1].Type,CustomEvent[1].Msg,CustomEvent[1].Comment);
	END_IF

	// Change sample variable randomly to trigger a value change event
	IF VariableMonitorExample = 0 THEN
		VariableMonitorExample := 10.5;
	END_IF

	// Error reset
	IF NOT MpAuditTrailSys.Error THEN
		MpAuditTrailSys.ErrorReset := FALSE;
	END_IF

	// Assign MpLinks & address references
	MpAuditTrailSys.MpLink := ADR(gMpLinkAuditTrail);
	MpAuditTrailSys.DeviceName := ADR('mappAuditFiles');
	MpAuditTrailConfigSys.MpLink := ADR(gMpLinkAuditTrail);
	MpAuditTrailConfigSys.Configuration := ADR(AuditTrailConfig);
	MpAuditTrailCEvents.MpLink := ADR(gMpLinkCustomEvents);
	MpAuditTrailUISys.MpLink := ADR(gMpLinkAuditTrail);
	MpAuditTrailUISys.UIConnect := ADR(MpAuditTrailUIConnect);

	// Call function blocks
	MpAuditTrailSys();
	MpAuditTrailConfigSys();
	MpAuditTrailCEvents();
	MpAuditTrailUISys();

	MpAuditTrailCEventsUI();
	MpAuditTrailCEvents();
	MpAuditTrailCEventsUI();

END_PROGRAM

PROGRAM _EXIT

	// Disable the function blocks to unlink the MpLinks
	MpAuditTrailSys.Enable := FALSE;
	MpAuditTrailConfigSys.Enable := FALSE;
	MpAuditTrailCEvents.Enable := FALSE;
	MpAuditTrailUISys.Enable := FALSE;

	// Call function blocks
	MpAuditTrailSys();
	MpAuditTrailConfigSys();
	MpAuditTrailCEvents();
	MpAuditTrailUISys();

END_PROGRAM
```

#### ChangeConfiguration.st
```iecst
ACTION ChangeConfiguration:

	MpAuditTrailConfigSys.MpLink := ADR(gMpLinkAuditTrail);
	MpAuditTrailConfigSys.Configuration := ADR(AuditTrailConfig);

	IF (MpAuditTrailConfigSys.Error) THEN
		IF (MpAuditTrailConfigSys.StatusID = mpAUDIT_ERR_CONFIG_LOAD) THEN
			LoadAuditConfiguration;
		END_IF
		MpAuditTrailConfigSys.Load := FALSE;
		MpAuditTrailConfigSys.Save := FALSE;
		MpAuditTrailConfigSys.ErrorReset := TRUE;
	END_IF

	MpAuditTrailConfigSys();
	MpAuditTrailConfigSys.ErrorReset := FALSE;

	IF (MpAuditTrailConfigSys.CommandDone) THEN
		IF (MpAuditTrailConfigSys.Load) THEN
			LoadAuditConfiguration;
		END_IF
		// after save the AuditTrail needs to restart
		IF (MpAuditTrailConfigSys.Save) THEN
			MpAuditTrailSys.Enable := FALSE;
		END_IF
		MpAuditTrailConfigSys.Load := FALSE;
		MpAuditTrailConfigSys.Save := FALSE;
	END_IF

END_ACTION
```

#### ExecuteQuery.st
```iecst
ACTION ExecuteQuery:

	// Initialize mapp function block
	QueryUserEvents.MpLink := ADR(gMpLinkAuditTrail);
	QueryUserEvents.Enable := TRUE;
	QueryUserEvents.Name := ADR(HmiAudit.Status.Query.Name);
	QueryUserEvents.Language := ADR('en');
	QueryUserEvents();

	CASE (AuditQuery.State) OF
		ACTIVE_AUDIT_WAIT:
			// Wait until the RunQuery command is triggered from the HMI.
			// If you prefer that the query runs anytime new data is available, then uncomment line 15 and comment out line 16 and delete
			// the "Run query" button from the HMI.
			//IF (AuditQuery.LastUpdateCount <> AuditQuery.UpdateCount) THEN
			IF (HmiAudit.Commands.RunQuery) THEN
				// Call the custom event function when the query execution is triggered
				MpAuditCustomEvent(gMpLinkCustomEvents,CustomEvent[2].Type,CustomEvent[2].Msg,CustomEvent[2].Comment);
				brsmemset(ADR(AuditQuery.Audits[0]), 0, SIZEOF(AuditQuery.Audits));
				AuditQuery.LastUpdateCount := AuditQuery.UpdateCount;
				QueryUserEvents.Execute := TRUE;
				HmiAudit.Commands.RunQuery := FALSE;
				IF (HmiAudit.Status.Query.Name = 'UserEvents') THEN
					HmiAudit.Status.Query.Option := 0;
				ELSIF (HmiAudit.Status.Query.Name = 'RecipeEvents') THEN
					HmiAudit.Status.Query.Option := 1;
				END_IF

				AuditQuery.State := ACTIVE_AUDIT_QUERY;
			END_IF

		ACTIVE_AUDIT_QUERY:
			// If the number of query results is less than MAX_QUERY_RESULTS, return to the wait state
			IF ((QueryUserEvents.CommandDone) AND (NOT QueryUserEvents.Info.HasMoreRows)) THEN
				// Call the custom event function when the query execution is done
				MpAuditCustomEvent(gMpLinkCustomEvents,"Cmd Done","Executing the query command has finished","For additional information check the logger.");
				QueryUserEvents.Execute := FALSE;
				QueryUserEvents.Next := FALSE;
				AuditQuery.State := ACTIVE_AUDIT_WAIT;
				// If the number of query results is more than MAX_QUERY_RESULTS, then query the next set of results
			ELSIF ((QueryUserEvents.CommandDone) AND (QueryUserEvents.Info.HasMoreRows)) THEN
				QueryUserEvents.Next := FALSE;
				AuditQuery.State := ACTIVE_AUDIT_NEXT;
			END_IF

		ACTIVE_AUDIT_NEXT:
			IF (AuditQuery.Next) THEN
				// By default, AuditQuery.Alarms has 20 elements, so it can hold 20 query results at a time (MAX_QUERY_RESULTS = 19).
				// If AuditQuery.Next is true, this means the query result is more than 20 alarms.
				// If you want to save the data for the first 20 alarms, add code here to copy AuditQuery.Alarms to another location.
				// Otherwise, the older alarms in the query will get overwritten with the newest entries here.
				brsmemset(ADR(AuditQuery.Audits[0]), 0, SIZEOF(AuditQuery.Audits));
				AuditQuery.Next := FALSE;
				QueryUserEvents.Next := TRUE;
				AuditQuery.State := ACTIVE_AUDIT_QUERY;
			END_IF
	END_CASE

	// Convert the query results into arrays that can easily be bound to the Table widget in mapp View
	FOR i := 0 TO MAX_QUERY_RESULTS DO
		HmiAudit.Status.Query.EvTime[i] := AuditQuery.Audits[i].EvTime;
		HmiAudit.Status.Query.Op[i] := AuditQuery.Audits[i].Op;
		HmiAudit.Status.Query.Text[i] := AuditQuery.Audits[i].Text;
		HmiAudit.Status.Query.DText[i] := AuditQuery.Audits[i].DText;
		HmiAudit.Status.Query.EvTimeString[i] := DT_TO_STRING(HmiAudit.Status.Query.EvTime[i]);
		IF HmiAudit.Status.Query.Text[i] <> "" THEN
			HmiAudit.Status.Query.EvTimeString[i] := RIGHT(HmiAudit.Status.Query.EvTimeString[i], 19);
		ELSE
			HmiAudit.Status.Query.EvTimeString[i] := '';
		END_IF;
	END_FOR

	// VC4
	IF HmiAudit.Status.Query.DPSelectedIndex = 0 THEN
		HmiAudit.Status.Query.Name := 'UserEvents';
	ELSIF HmiAudit.Status.Query.DPSelectedIndex = 1 THEN
		HmiAudit.Status.Query.Name := 'RecipeEvents';
	END_IF;
	HmiAudit.Status.ArchiveSetupVisibility := NOT HmiAudit.Status.ArchiveAvailable;
	HmiAudit.Status.ArchiveSetupTimeOfDayVisibility := (HmiAudit.Parameters.ArchiveSettings.Mode = mpAUDIT_ARCHIVE_BATCH);

END_ACTION
```

#### HMIActions.st
```iecst
ACTION ArchiveExport:

	// Assign variables to exchange with the HMI
	MpAuditTrail_0.ExportArchive := HmiAudit.Commands.ExportArchives;
	HmiAudit.Status.ArchiveAvailable := MpAuditTrail_0.ArchiveAvailable;
	HmiAudit.Status.NumberOfArchives := MpAuditTrail_0.Info.NumberArchives;

	IF (HmiAudit.Commands.ExportArchives AND MpAuditTrail_0.CommandDone) THEN
		HmiAudit.Commands.ExportArchives := FALSE;
	END_IF

END_ACTION

ACTION ArchiveSettings:

	// Audit Trail Config implementation
	IF (HmiAudit.Commands.SaveConfig = TRUE) THEN
		HmiAudit.Commands.SaveConfig := FALSE;
		SaveAuditConfiguration;
		MpAuditTrailConfig_0.Save := TRUE;
	END_IF

	// After the configuration has been changed the AuditTrail is reset (disabled). This re-enables the component
	IF MpAuditTrail_0.Active = FALSE THEN
		MpAuditTrail_0.Enable := TRUE;
	END_IF

END_ACTION

ACTION SaveAuditConfiguration:

	// Assign current parameters from the HMI structure to AuditTrail configuration before saving it
	AuditTrailConfig.Archive.Time := UDINT_TO_TOD((((USINT_TO_UDINT(HmiAudit.Parameters.ArchiveSettings.Hour) * 60) +
	HmiAudit.Parameters.ArchiveSettings.Minute) * 60) * 1000);
	AuditTrailConfig.Archive.Enable := HmiAudit.Parameters.ArchiveSettings.Enable;
	AuditTrailConfig.Archive.MaxSize := HmiAudit.Parameters.ArchiveSettings.MaxSize;
	AuditTrailConfig.Archive.Mode := HmiAudit.Parameters.ArchiveSettings.Mode;
	AuditTrailConfig.Export.FileType := HmiAudit.Parameters.ArchiveSettings.FileType;

	// Save current archive setings to retain variable
	ArchiveSettingsRetain := HmiAudit.Parameters.ArchiveSettings;

 END_ACTION

ACTION LoadAuditConfiguration:

	// Assign current parameters from the configuration to the HMI structure
	HmiAudit.Parameters.ArchiveSettings.Hour := UDINT_TO_USINT(TOD_TO_UDINT(AuditTrailConfig.Archive.Time) / 1000 / 60 / 60);
	HmiAudit.Parameters.ArchiveSettings.Minute := UDINT_TO_USINT(TOD_TO_UDINT(AuditTrailConfig.Archive.Time) / 1000 / 60) -
													(HmiAudit.Parameters.ArchiveSettings.Hour * 60);
	HmiAudit.Parameters.ArchiveSettings.Enable := AuditTrailConfig.Archive.Enable;
	HmiAudit.Parameters.ArchiveSettings.MaxSize := AuditTrailConfig.Archive.MaxSize;
	HmiAudit.Parameters.ArchiveSettings.Mode := AuditTrailConfig.Archive.Mode;
	HmiAudit.Parameters.ArchiveSettings.FileType := AuditTrailConfig.Export.FileType;

END_ACTION

ACTION QueryTableConfig:

	// Configure visible list
	HmiAudit.Status.TableConfig[0] := '{ "specRows": [{"from":';
	HmiAudit.Status.Query.QueryCount := 0;
	FOR i := 0 TO 9 DO
		IF HmiAudit.Status.Query.Text[i] <> "" THEN
			HmiAudit.Status.Query.QueryCount := i + 1;
		END_IF
	END_FOR
	brsitoa((HmiAudit.Status.Query.QueryCount), ADR(HmiAudit.Status.TableConfig[0]) + brsstrlen(ADR(HmiAudit.Status.TableConfig[0])));
	brsstrcat(ADR(HmiAudit.Status.TableConfig[0]), ADR(',"to":19, "visible":false}]'));

	// Hide operator column for the recipe query
	IF (HmiAudit.Status.Query.Option = 0) THEN
		brsstrcat(ADR(HmiAudit.Status.TableConfig[0]), ADR(', "specColumns": [ {"from":1, "to":1, "visible":true}]'));
	ELSIF (HmiAudit.Status.Query.Option = 1) THEN
		brsstrcat(ADR(HmiAudit.Status.TableConfig[0]), ADR(', "specColumns": [ {"from":1, "to":1, "visible":false}]'));
	END_IF

	brsstrcat(ADR(HmiAudit.Status.TableConfig[0]), ADR('}'));

END_ACTION
```


### Package Logical/Infrastructure/VC4/Report - Package for mapp Report Framework

### Program Logical/Infrastructure/VC4/Report/ReportMgr

#### ReportMgr.typ
```iecst
(*Structure types*)

TYPE
	ReportHmiInterfaceType : 	STRUCT
		Commands : ReportCommandsType; (*Structure to hold the commands from the HMI*)
		Parameters : ReportParametersType; (*Structure to hold the parameters from the HMI*)
		Status : ReportStatusType; (*Structure to hold the status information from the HMI*)
	END_STRUCT;
	ReportCommandsType : 	STRUCT  (*Structure to hold the commands from the HMI*)
		Generate : BOOL; (*Generate a report*)
		Reset : BOOL; (*Reset the report function block*)
	END_STRUCT;
	ReportParametersType : 	STRUCT  (*Structure to hold the parameters from the HMI*)
		Name : STRING[50]; (*Name of the report*)
		UseAdvancedFormat : BOOL; (*Whether or not the report should use the advanced format*)
		PathOfReportToView : STRING[255]; (*The file path of the selected report*)
		SelectedLanguage : STRING[10] := 'en'; (*Selected language*)
	END_STRUCT;
	ReportStatusType : 	STRUCT  (*Structure to hold the status information from the HMI*)
		ViewAllowed : BOOL; (*Bit to indicate it is allowable to view a report right now*)
		DeleteAllowed : BOOL; (*Bit to indicate it is allowable to delete a report right now*)
		CreateAllowed : BOOL; (*Bit to indicate it is allowable to create a report right now*)
		Busy : BOOL; (*Report is busy executing an action*)
		Error : BOOL; (*Error flag*)
		CurrentFormat : ReportFormatEnum; (*Current report format*)
		FileOverMax : BOOL; (*Active when more than 50 items detected*)
		FileNames : ARRAY[0..49]OF STRING[50]; (*Existing report file names*)
		TempFilePath : ARRAY[0..49]OF STRING[255]; (*A temporary variable used to concatonate and build the full file path of the selected file*)
		FilePath : ARRAY[0..49]OF STRING[255]; (*The full file path of the selcted file*)
		TimeStamps : ARRAY[0..49]OF DATE_AND_TIME; (*Time stamps for existing reports*)
		TimeStampsText : ARRAY[0..49]OF STRING[80]; (*Time stamps for existing reports*)
		Size : {REDUND_UNREPLICABLE} ARRAY[0..49]OF UDINT; (*Sizes of existing report files*)
		SelectedIndex : USINT; (*Index of the selected file*)
		LastSelectedIndex : USINT := 255; (*Index of the last selected report file*)
		LastSelectedDeviceIndex : UINT; (*Index of the last selected file device. Compared with MpFileManagerUIConnect.DeviceList.SelectedIndex*)
		TableConfig : ARRAY[0..1]OF STRING[120]; (*Table configuration for the list of available reports*)
		FilterString : STRING[1000]; (*String used to filter out any file that is not a PDF*)
		Layer : ReportStatusLayerType;
		PageUpDownVisibility : USINT;
	END_STRUCT;
	ReportExampleType : 	STRUCT  (*Structure for the example data used by the two types of reports*)
		SimpleReport : SimpleReportDataType; (*Structure for the simple report's example data*)
		AdvancedReport : AdvReportDataType; (*Structure for the advanced report's example data*)
	END_STRUCT;
	AdvReportDataType : 	STRUCT  (*Structure to hold a report's advanced example data*)
		OeeLine : ARRAY[0..NUM_LINES]OF ReportDataOeeType := [(RunTime:=T#24h00m00s00ms,UpTime:=T#23h13m34s98ms,DownTime:=T#00h47m25s02ms,PartsMade:=67268,PPM:=46.7138,NumRejects:=1256,TemperatureSample:=(Value:=[99,97,103,101,100,102,95,2(105),100,102,101,96,105,3(20),97,100,96,99,105,101,97,2(103),98,100,99,104,100,105,104,99,104,103,104,102,100,101,102,96,105,99,97,100,103,105,102,101,97,105,95,101,2(103),2(101),100,101,99,105,101,102,96,95,100,98,103,105,99,104,96,97,96,101,103,100,103,95,102,97,105,103,99,96,98,105,95,103,100,103,100,2(105),101])),(RunTime:=T#24h00m00s00ms,UpTime:=T#23h54m09s00ms,DownTime:=T#00h05m51s00ms,PartsMade:=75061,PPM:=52.1256,NumRejects:=805,TemperatureSample:=(Value:=[98,104,103,97,98,95,101,97,104,96,100,101,103,105,95,103,2(96),98,104,97,102,100,2(96),102,101,95,104,99,104,96,99,104,96,101,105,98,101,99,105,100,97,2(101),96,101,2(100),99,96,101,100,105,97,100,101,99,97,99,104,105,102,97,105,104,98,102,103,102,98,105,103,100,99,104,101,99,105,100,105,102,99,2(95),103,96,97,95,100,99,96,102,105,95,96])),(RunTime:=T#24h00m00s00ms,UpTime:=T#15h57m16s13ms,DownTime:=T#08h02m43s87ms,PartsMade:=40235,PPM:=27.9409,NumRejects:=742,TemperatureSample:=(Value:=[2(97),100,105,104,101,105,97,103,16(20),96,103,100,101,99,102,95,99,102,99,103,95,102,99,96,2(102),103,2(99),102,3(97),101,105,103,2(101),104,101,104,105,97,100,2(99),100,103,101,103,95,103,96,100,99,20(20),99,96,95,96,98]))]; (*Structure to hold example data of a line's OEE statistics*)
		BatchNumber : UDINT := 23561458; (*An example of a batch number used for an advanced report*)
	END_STRUCT;
	SimpleReportDataType : 	STRUCT  (*Structure to hold a report's example data*)
		OeeLine : ARRAY[0..NUM_LINES]OF ReportDataOeeType := [(RunTime:=T#24h00m00s00ms,UpTime:=T#23h13m34s98ms,DownTime:=T#00h47m25s02ms,PartsMade:=67268,PPM:=46.7138,NumRejects:=1256,TemperatureSample:=(Value:=[99,97,103,101,100,102,95,2(105),100,102,101,96,105,3(20),97,100,96,99,105,101,97,2(103),98,100,99,104,100,105,104,99,104,103,104,102,100,101,102,96,105,99,97,100,103,105,102,101,97,105,95,101,2(103),2(101),100,101,99,105,101,102,96,95,100,98,103,105,99,104,96,97,96,101,103,100,103,95,102,97,105,103,99,96,98,105,95,103,100,103,100,2(105),101])),(RunTime:=T#24h00m00s00ms,UpTime:=T#23h54m09s00ms,DownTime:=T#00h05m51s00ms,PartsMade:=75061,PPM:=52.1256,NumRejects:=805,TemperatureSample:=(Value:=[98,104,103,97,98,95,101,97,104,96,100,101,103,105,95,103,2(96),98,104,97,102,100,2(96),102,101,95,104,99,104,96,99,104,96,101,105,98,101,99,105,100,97,2(101),96,101,2(100),99,96,101,100,105,97,100,101,99,97,99,104,105,102,97,105,104,98,102,103,102,98,105,103,100,99,104,101,99,105,100,105,102,99,2(95),103,96,97,95,100,99,96,102,105,95,96])),(RunTime:=T#24h00m00s00ms,UpTime:=T#15h57m16s13ms,DownTime:=T#08h02m43s87ms,PartsMade:=40235,PPM:=27.9409,NumRejects:=742,TemperatureSample:=(Value:=[2(97),100,105,104,101,105,97,103,16(20),96,103,100,101,99,102,95,99,102,99,103,95,102,99,96,2(102),103,2(99),102,3(97),101,105,103,2(101),104,101,104,105,97,100,2(99),100,103,101,103,95,103,96,100,99,20(20),99,96,95,96,98]))]; (*Structure to hold example data of a line's OEE statistics*)
	END_STRUCT;
	ReportDataOeeType : 	STRUCT  (*Structure to hold example data of a line's OEE statistics*)
		RunTime : TIME; (*How long the line has been running*)
		UpTime : TIME; (*How long the line has been up*)
		DownTime : TIME; (*How long the line has been down*)
		PartsMade : UDINT; (*How many parts the line has made*)
		PPM : REAL; (*The average parts per minute made by the line*)
		NumRejects : UDINT; (*The number of rejected parts made by the line*)
		TemperatureSample : ReportDataTempSampleType; (*Temperature samples from the line*)
	END_STRUCT;
	ReportDataTempSampleType : 	STRUCT  (*Temperature samples from the line*)
		TimeStamp : ARRAY[0..NUM_TEMP_SAMPLES]OF INT; (*The time the temperature sample was taken*)
		Value : ARRAY[0..NUM_TEMP_SAMPLES]OF REAL; (*The actual temperature reading*)
	END_STRUCT;
END_TYPE

(*Enumerations*)

TYPE
	ReportFormatEnum :
		( (*An enumeration of the format selected by the user for the report*)
		FORMAT_SIMPLE, (*A simple report to showcase some features of mapp Report*)
		FORMAT_ADVANCED (*An advanced report to showcase some features of mapp Report*)
		);
END_TYPE

(**)

TYPE
	ReportStatusLayerType : 	STRUCT
		ReportCreate : USINT;
		ReportDelete : USINT;
		ReportView : USINT;
	END_STRUCT;
END_TYPE

(**)
(**)

TYPE
	HtmlViewType : 	STRUCT
		HTMLStream : STRING[255];
		ChangeURLDatapoint : STRING[255];
		CurrentURLDatapoint : STRING[255];
	END_STRUCT;
END_TYPE
```

#### ReportMgr.var
```iecst
(*Function Blocks*)
VAR
	MpReportCoreSys : MpReportCore; (*MpReport instance*)
	MpFileManagerUIReport : MpFileManagerUI; (*MpFileManagerUI instance*)
	DirCreateReport : DirCreate; (*DirCreate instance*)
END_VAR
(*Constants*)
VAR CONSTANT
	NUM_LINES : INT := 2; (*The number lines on the machine*)
	NUM_TEMP_SAMPLES : INT := 95; (*The number of temperature samples in the example data*)
END_VAR
(*Structure Types*)
VAR
	HmiReport : ReportHmiInterfaceType; (*HMI interface structure*)
	ReportExample : ReportExampleType; (*Structure for the example data used by the two types of reports*)
	MpFileManagerUIConnect : MpFileManagerUIConnectType := (DeviceList:=(DeviceNames:=['mappReportFiles',9('')])); (*MpFile connection to the HMI*)
END_VAR
(*Variables*)
VAR
	i : USINT; (*Index*)
	TimeIndex : INT; (*Index to loop through file devices*)
	tempDeviceIndex : USINT; (*Temporary index for identifying USB devices*)
	ItemCount : UDINT; (*Counter for available files*)
END_VAR
```
